(* IEC 61131-3 sources: SmartHomeNew/snapshots/2026-05-25, 217 files *)

(* ---- E_ALERT_PRIORITY.dut ---- *)
{attribute 'strict'}
TYPE E_ALERT_PRIORITY :
(
    ALERT_PRIORITY_NONE := 0,
    ALERT_PRIORITY_LOW := 1,
    ALERT_PRIORITY_MEDIUM := 2,
    ALERT_PRIORITY_HIGH := 3,
    ALERT_PRIORITY_CRITICAL := 4
) USINT;
END_TYPE

(* ---- E_Modbus_Function.dut ---- *)
TYPE E_Modbus_Function :
(
    MB_NONE := 0,
    MB_FC03_READ_HOLDING_REGISTERS := 3,
    MB_FC04_READ_INPUT_REGISTERS := 4,
    MB_FC06_WRITE_SINGLE_REGISTER := 6,
    MB_FC16_WRITE_MULTIPLE_REGISTERS := 16
);
END_TYPE

(* ---- E_OpenTherm_Error.dut ---- *)
TYPE E_OpenTherm_Error :
(
    OT_ERROR_NONE := 0,
    OT_ERROR_HEARTBEAT_TIMEOUT := 1,
    OT_ERROR_ACK_TIMEOUT := 2,
    OT_ERROR_ADAPTER_FAULT := 3,
    OT_ERROR_COMMUNICATION := 4,
    OT_ERROR_INVALID_RESPONSE := 5
);
END_TYPE

(* ---- E_Rule_Condition_Type.dut ---- *)
{attribute 'strict'}
TYPE E_Rule_Condition_Type :
(
    COND_NONE := 0,
    COND_AIR_TEMP := 1,
    COND_FLOOR_TEMP := 2,
    COND_HUMIDITY := 3,
    COND_CO2 := 4,
    COND_METHANE := 5,
    COND_CO := 6,
    COND_DOOR_WINDOW := 7,
    COND_FLOOD := 8,
    COND_SMOKE := 9,
    COND_MOTION := 10,
    COND_TIME_OF_DAY := 11,
    COND_DAY_OF_WEEK := 12
) USINT;
END_TYPE

(* ---- E_RUNTIME_ADAPTIVE_MODE.dut ---- *)
TYPE E_RUNTIME_ADAPTIVE_MODE : (
    FULL_SEMANTIC_MODE,
    REDUCED_ANALYTICS_MODE,
    SURVIVABILITY_MODE,
    MINIMAL_SAFE_MODE
);
END_TYPE

(* ---- E_RUNTIME_TRANSITION_RESULT.dut ---- *)
TYPE E_RUNTIME_TRANSITION_RESULT : (
    TRANSITION_VALID,
    TRANSITION_FORBIDDEN,
    TRANSITION_REQUIRES_PROOF,
    TRANSITION_REQUIRES_RECOVERY,
    TRANSITION_REQUIRES_TEMPORAL_ALIGNMENT
);
END_TYPE

(* ---- E_SCENARIO_TYPE.dut ---- *)
{attribute 'strict'}
TYPE E_SCENARIO_TYPE :
(
    SCENARIO_NONE := 0,
    SCENARIO_MORNING := 1,
    SCENARIO_EVENING := 2,
    SCENARIO_AWAY := 3,
    SCENARIO_PARTY := 4,
    SCENARIO_SLEEP := 5,
    SCENARIO_EMERGENCY := 6,
    SCENARIO_PRESENCE := 7
) USINT;
END_TYPE

(* ---- GVL_CANONICAL_RUNTIME_FABRIC_REGISTRY.gvl ---- *)
TYPE E_GOVERNANCE_PRIORITY_TIER : (
    TIER_0_SAFETY,
    TIER_1_AUTHORITY,
    TIER_2_PHYSICAL_TRUTH,
    TIER_3_SURVIVABILITY,
    TIER_4_OBSERVABILITY,
    TIER_5_ANALYTICS
);
END_TYPE

VAR_GLOBAL
    // Canonical semantic registry.
    Runtime_Fabric_Registry_Active : BOOL := TRUE;
    Runtime_Fabric_Registry_ReadOnly : BOOL := TRUE;

    // Tier hierarchy.
    Current_Governance_Priority_Tier : E_GOVERNANCE_PRIORITY_TIER := TIER_0_SAFETY;

    Tier0_Safety_Active : BOOL := TRUE;
    Tier1_Authority_Active : BOOL := TRUE;
    Tier2_Physical_Truth_Active : BOOL := TRUE;
    Tier3_Survivability_Active : BOOL := TRUE;
    Tier4_Observability_Active : BOOL := TRUE;
    Tier5_Analytics_Active : BOOL := TRUE;

    // Canonical semantic domains.
    Temporal_Integrity_Cluster_Active : BOOL := TRUE;
    Authority_Integrity_Cluster_Active : BOOL := TRUE;
    Physical_Reality_Cluster_Active : BOOL := TRUE;
    Operational_Intelligence_Cluster_Active : BOOL := TRUE;
    Survivability_Cluster_Active : BOOL := TRUE;

    // Runtime compression observations.
    Governance_Scattering_Observed : BOOL := FALSE;
    Semantic_Duplication_Observed : BOOL := FALSE;
    Runtime_Complexity_Pressure_Observed : BOOL := FALSE;

    // Semantic recursion prevention.
    Governance_Depth_Limit_Reached : BOOL := FALSE;
    Semantic_Recursion_Limit_Reached : BOOL := FALSE;
    Verification_Chaining_Limit_Reached : BOOL := FALSE;
    Observability_Amplification_Limit_Reached : BOOL := FALSE;

    // Runtime cost awareness.
    Governance_Runtime_Cost_Observed : BOOL := FALSE;
    Verification_Induced_Instability_Risk : BOOL := FALSE;

    Runtime_Fabric_Registry_Epoch : UDINT := 0;
END_VAR

(* ---- ST_Alarm_Record.dut ---- *)
{attribute 'pack_mode' := '1'}
TYPE ST_Alarm_Record :
STRUCT
    ID : UDINT; // Уникальный идентификатор тревоги
    Timestamp_MS : UDINT; // Время возникновения
    Source : STRING(20); // Источник (Gas, Fire, Flood, Security, System)
    Source_ID : BYTE; // Идентификатор источника (например, номер котла)
    Message : STRING(100); // Описание тревоги
    Severity : E_ALERT_PRIORITY; // Приоритет тревоги
    Is_Active : BOOL; // Тревога все еще активна
    Is_Acknowledged : BOOL; // Квитирована оператором
END_STRUCT
END_TYPE

(* ---- ST_Behavior_Weights.dut ---- *)
TYPE ST_Behavior_Weights :
STRUCT
    W_Comfort : REAL;
    W_Night : REAL;
    W_Preheat : REAL;
    W_VentBoost : REAL;
    W_AccessSecure : REAL;
END_STRUCT
END_TYPE

(* ---- ST_Calibration_Sensor_Summary.dut ---- *)
{attribute 'pack_mode' := '1'}
TYPE ST_Calibration_Sensor_Summary :
STRUCT
    active : BOOL;
    status : INT; // 0=OK,1=IN_PROGRESS,2=WARNING,3=ERROR
    calibrated_value : REAL;
    deviation_percent : REAL;
    verification_active : BOOL;
    verification_failed : BOOL;
    record_index : INT;
    label : STRING(64);
    summary_text : STRING(160);
END_STRUCT
END_TYPE

(* ---- ST_Distributed_Authority_State.dut ---- *)
TYPE ST_Distributed_Authority_State :
STRUCT
    Runtime_Valid : BOOL;
    Runtime_System_Time_MS : UDINT;

    Controller_Id : UINT;
    Runtime_Node_Id : UINT;
    Authority_Domain_Id : UINT;

    Authority_Election_Active : BOOL;
    Authority_Master_Elected : BOOL;
    Authority_Backup_Elected : BOOL;
    Authority_Observer_Only : BOOL;

    Authority_Lease_Valid : BOOL;
    Authority_Lease_Expired : BOOL;
    Authority_Lease_Timeout_MS : UDINT;

    Replication_Consensus_Healthy : BOOL;
    Replication_Consensus_Stale : BOOL;

    Recovery_Authority_Allowed : BOOL;
    Rollback_Authority_Allowed : BOOL;
    Quarantine_Authority_Allowed : BOOL;

    Split_Brain_Blocked : BOOL;
    Distributed_Safety_Barrier_OK : BOOL;

    Status_Code : UINT;
    Status_Text : STRING(160);
END_STRUCT
END_TYPE

(* ---- ST_Distributed_Orchestration_State.dut ---- *)
TYPE ST_Distributed_Orchestration_State :
STRUCT
    Runtime_Valid : BOOL;
    Runtime_System_Time_MS : UDINT;

    Orchestration_Sequence_Id : UDINT;
    Distributed_Execution_Active : BOOL;

    Cross_Node_Isolation_Required : BOOL;
    Cross_Node_Recovery_Required : BOOL;
    Cross_Node_Rollback_Required : BOOL;

    Distributed_Projection_Granted : BOOL;
    Distributed_Projection_Blocked : BOOL;

    Distributed_Rollback_Allowed : BOOL;
    Distributed_Recovery_Allowed : BOOL;

    Distributed_Scheduler_Healthy : BOOL;
    Distributed_Timing_Window_Valid : BOOL;

    Remote_Node_Ack_Required : BOOL;
    Remote_Node_Ack_Received : BOOL;

    Distributed_Conflict_Detected : BOOL;
    Distributed_Split_Execution_Suspected : BOOL;

    Status_Code : UINT;
    Status_Text : STRING(160);
END_STRUCT
END_TYPE

(* ---- ST_Flood_Global_Config.dut ---- *)
{attribute 'pack_mode' := '1'}
TYPE ST_Flood_Global_Config :
STRUCT
    // Isolation groups:
    // 1 = стояк 1 кухня, 2 = стояк 2 мастер-санузел,
    // 3 = стояк 3 гостевые санузлы + постирочная,
    // 4 = общий ввод ХВС/ГВС, legacy chains 35/36.
    // Вода от скважины: при потере питания насос останавливается и давления нет,
    // поэтому базовая эксплуатационная модель — нормально-открытые краны с
    // электроприводом и концевиками, закрываемые при аварии.
    valve_types : ARRAY[1..GVL_CONSTANTS.C_MAX_FLOOD_VALVES] OF E_VALVE_TYPE := [GVL_CONSTANTS.C_MAX_FLOOD_VALVES(E_VALVE_TYPE.VALVE_NO)];

    // 1-2 кухня -> стояк 1;
    // 3-4 мастер-санузел -> стояк 2;
    // 5-9 гостевые санузлы + постирочная -> стояк 3;
    // 10-12 котельная/ХВП/общий ввод -> общий ввод 35/36.
    sensor_to_valve_map : ARRAY[1..GVL_CONSTANTS.C_MAX_FLOOD_SENSORS] OF BYTE := [1, 1, 2, 2, 3, 3, 3, 3, 3, 4, 4, 4];

    min_duration_ms : UDINT := 5000; // Защита от брызг (5 сек)
    warning_duration_ms : UDINT := 30000; // Время предупреждения до перекрытия (30 сек)
END_STRUCT
END_TYPE

(* ---- ST_FloorHeating_Circuit_Config.dut ---- *)
{attribute 'pack_mode' := '1'}
TYPE ST_FloorHeating_Circuit_Config :
STRUCT
    circuit_id : BYTE := 0;
    zone : BYTE := 0;
    manifold_id : BYTE := 1; // ID коллектора, к которому подключен контур
    sensor_id : BYTE := 1; // ID датчика температуры
    valve_id : BYTE := 1; // ID клапана
    control_type : BYTE := 1; // 0: по полу, 1: по воздуху

    // Legacy/default setpoint. Kept for backward compatibility.
    // If comfort_temp <= 0.0, design_temp remains the comfort setpoint.
    design_temp : REAL := 35.0;

    // Per-room/per-circuit comfort and economy policy.
    // use_in_normal=FALSE keeps the circuit at economy_temp even in normal mode.
    // use_in_away_preheat=TRUE allows planned-return preheat to comfort_temp.
    use_in_normal : BOOL := TRUE;
    use_in_away_preheat : BOOL := TRUE;
    comfort_temp : REAL := 0.0; // 0.0 = use design_temp
    economy_temp : REAL := 16.0;
    long_away_temp : REAL := 12.0;

    min_temp : REAL := 20.0;
    max_temp : REAL := 45.0;
    pid_kp : REAL := 2.0;
    pwm_period_s : UINT := 600; // Период ШИМ в секундах (по умолчанию 10 минут)
END_STRUCT
END_TYPE

(* ---- ST_Forensic_Journal_Record.dut ---- *)
TYPE ST_Forensic_Journal_Record :
STRUCT
    Record_Valid : BOOL;
    Event_Time_MS : UDINT;
    Event_Id : UDINT;
    Event_Class : UINT;
    Event_Severity : UINT;

    Config_Version : UDINT;
    Topology_Version : UDINT;
    Recovery_Domain_Id : UINT;
    Valve_Group_Id : UINT;
    Sensor_Id : UINT;

    Activation_Event : BOOL;
    Rollback_Event : BOOL;
    Quarantine_Event : BOOL;
    Recovery_Event : BOOL;
    Restart_Event : BOOL;

    Status_Code : UINT;
    Event_Text : STRING(160);
END_STRUCT
END_TYPE

(* ---- ST_Heating_Circuit_Runtime_Projection.dut ---- *)
TYPE ST_Heating_Circuit_Runtime_Projection :
STRUCT
    // Passive runtime-to-observability projection contract.
    // Contains semantic runtime state only.
    // No runtime authority.

    Visible : BOOL;

    // Selected operational source
    Selected_Source_Code : UINT; // 0 none, 1 room, 2 floor
    Selected_Source_Confidence : REAL;

    // Runtime degraded semantics
    Fallback_Active : BOOL;
    Source_Degraded : BOOL;
    Sensor_Error_Active : BOOL;

    // Explainability semantics
    Reason_Code : UINT;
    Reason_Text : STRING(128);

    // Runtime semantic edge publication
    Source_Switched_Event : BOOL;
    Fallback_Activated_Event : BOOL;
    Fallback_Recovered_Event : BOOL;
    Source_Loss_Event : BOOL;

    Last_Event_Code : UINT;
    Last_Event_Text : STRING(128);
    Last_Event_MS : UDINT;
END_STRUCT
END_TYPE

(* ---- ST_Heating_Runtime_Blackbox_Timeline.dut ---- *)
TYPE ST_Heating_Runtime_Blackbox_Timeline :
STRUCT
    // ======================================================
    // Blackbox events
    // ======================================================
    Events : ARRAY[1..256] OF ST_Heating_Runtime_Blackbox_Event;

    // ======================================================
    // Timeline state
    // ======================================================
    Write_Index : UINT;
    Event_Count : UINT;
    Timeline_Overflow : BOOL;

    // ======================================================
    // Runtime forensic state
    // Passive forensic visibility only.
    // No replay activation authority exists.
    // ======================================================
    Reconstruction_Visible : BOOL;
    Forensic_Timeline_Visible : BOOL;
    Root_Cause_Reconstructed : BOOL;

    // ======================================================
    // Timeline integrity
    // ======================================================
    Sequencing_Valid : BOOL;
    Ownership_Valid : BOOL;
    Synchronization_Valid : BOOL;

    // ======================================================
    // Timeline status
    // ======================================================
    Status_Code : UINT;
    Status_Text : STRING(128);
END_STRUCT
END_TYPE

(* ---- ST_Heating_Runtime_Context.dut ---- *)
TYPE ST_Heating_Runtime_Context :
STRUCT
    // ======================================================
    // Runtime lifecycle
    // ======================================================
    Runtime_Enabled : BOOL;
    Runtime_Ready : BOOL;
    Runtime_Fault : BOOL;

    // ======================================================
    // Runtime phase model
    // ======================================================
    Current_Phase : E_Heating_Runtime_Phase;

    // ======================================================
    // Phase execution permissions
    // ======================================================
    Allow_DHW_Phase : BOOL;
    Allow_Heating_Phase : BOOL;
    Allow_Service_Gating_Phase : BOOL;
    Allow_State_Publication_Phase : BOOL;
    Allow_Diagnostics_Phase : BOOL;
    Allow_Output_Projection_Phase : BOOL;

    // ======================================================
    // Runtime sequencing validation
    // ======================================================
    DHW_Executed : BOOL;
    Heating_Executed : BOOL;
    Service_Gating_Executed : BOOL;
    State_Publication_Executed : BOOL;
    Diagnostics_Executed : BOOL;
    Output_Projection_Executed : BOOL;

    // ======================================================
    // Runtime ordering integrity
    // ======================================================
    DHW_Before_Heating_Valid : BOOL;
    State_Publication_Before_Diagnostics_Valid : BOOL;
    Output_Projection_Last_Valid : BOOL;

    // ======================================================
    // Runtime status
    // ======================================================
    Runtime_Status_Code : UINT;
    Runtime_Status_Text : STRING(128);

    // ======================================================
    // Diagnostics / explainability isolation
    // ======================================================
    Diagnostics_Isolation_Valid : BOOL;
    Explainability_Isolation_Valid : BOOL;

    // ======================================================
    // Safety isolation
    // ======================================================
    Safety_Isolation_Valid : BOOL;

    // ======================================================
    // OpenTherm ownership isolation
    // ======================================================
    OpenTherm_Ownership_Valid : BOOL;

    // ======================================================
    // Cascade ownership isolation
    // ======================================================
    Cascade_Ownership_Valid : BOOL;
END_STRUCT
END_TYPE

(* ---- ST_Heating_Runtime_Observation.dut ---- *)
TYPE ST_Heating_Runtime_Observation :
STRUCT
    // ======================================================
    // Runtime execution state
    // ======================================================
    Runtime_Active : BOOL;
    Runtime_Ready : BOOL;
    Runtime_Fault : BOOL;

    // ======================================================
    // Runtime phase observation
    // ======================================================
    Current_Phase : E_Heating_Runtime_Phase;

    // ======================================================
    // DHW runtime observation
    // ======================================================
    DHW_Demand_Active : BOOL;
    DHW_Heating_Active : BOOL;
    DHW_Circulation_Active : BOOL;

    // ======================================================
    // Heating runtime observation
    // ======================================================
    Heating_Demand_Active : BOOL;
    Heating_Runtime_Active : BOOL;
    Heating_Output_Active : BOOL;

    // ======================================================
    // Cascade runtime observation
    // ======================================================
    Cascade_Available : BOOL;
    Cascade_Degraded : BOOL;
    Cascade_Active_Boilers : UINT;
    Cascade_Available_Boilers : UINT;

    // ======================================================
    // OpenTherm runtime observation
    // ======================================================
    OpenTherm_Online : BOOL;
    OpenTherm_Command_Valid : BOOL;
    OpenTherm_Transport_Degraded : BOOL;

    // ======================================================
    // Diagnostics observation
    // ======================================================
    Diagnostics_Active : BOOL;
    Explainability_Active : BOOL;

    // ======================================================
    // Runtime sequencing observation
    // ======================================================
    DHW_Before_Heating_Observed : BOOL;
    Diagnostics_After_Publication_Observed : BOOL;
    Output_Projection_Last_Observed : BOOL;

    // ======================================================
    // Runtime ownership observation
    // ======================================================
    Runtime_Ownership_Valid : BOOL;
    Diagnostics_Ownership_Valid : BOOL;
    OpenTherm_Ownership_Valid : BOOL;
    Cascade_Ownership_Valid : BOOL;
    Safety_Ownership_Valid : BOOL;

    // ======================================================
    // Runtime observation status
    // ======================================================
    Observation_Status_Code : UINT;
    Observation_Status_Text : STRING(128);
END_STRUCT
END_TYPE

(* ---- ST_Heating_Runtime_Phase_Transition.dut ---- *)
TYPE ST_Heating_Runtime_Phase_Transition :
STRUCT
    // ======================================================
    // Phase transition state
    // ======================================================
    Previous_Phase : E_Heating_Runtime_Phase;
    Current_Phase : E_Heating_Runtime_Phase;
    Next_Phase : E_Heating_Runtime_Phase;

    // ======================================================
    // Transition lifecycle
    // ======================================================
    Transition_Active : BOOL;
    Transition_Completed : BOOL;
    Transition_Failed : BOOL;

    // ======================================================
    // Transition timing
    // ======================================================
    Transition_Start_MS : UDINT;
    Transition_End_MS : UDINT;
    Transition_Duration_MS : UDINT;

    // ======================================================
    // Transition integrity
    // ======================================================
    Sequencing_Valid : BOOL;
    Ownership_Valid : BOOL;
    Synchronization_Valid : BOOL;

    // ======================================================
    // Transition status
    // ======================================================
    Status_Code : UINT;
    Status_Text : STRING(128);
END_STRUCT
END_TYPE

(* ---- ST_IO_Binding_Record.dut ---- *)
TYPE ST_IO_Binding_Record :
STRUCT
    Binding_Valid : BOOL;
    Binding_Version : UDINT;

    Physical_Channel_Id : UINT;
    Logical_Device_Id : UINT;
    Domain_Id : UINT;
    Role_Id : UINT;

    Controller_Id : UINT;
    Module_Id : UINT;
    Terminal_Id : UINT;

    Inverted : BOOL;
    Required : BOOL;
    Quality_Required : BOOL;

    Status_Code : UINT;
    Status_Text : STRING(128);
END_STRUCT
END_TYPE

(* ---- ST_Modbus_Request.dut ---- *)
TYPE ST_Modbus_Request :
STRUCT
    Enable : BOOL;
    Slave_ID : BYTE;
    Function_Code : E_Modbus_Function;
    Start_Register : UINT;
    Register_Count : UINT;
    Write_Value : ARRAY[1..32] OF WORD;
    Sequence : UDINT;
    Timeout_MS : UDINT;
END_STRUCT
END_TYPE

(* ---- ST_OpenTherm_Command.dut ---- *)
TYPE ST_OpenTherm_Command :
STRUCT
    Enable : BOOL;
    Setpoint_x10 : UINT;
    Sequence : UDINT;
    Last_Write_MS : UDINT;
END_STRUCT
END_TYPE

(* ---- ST_OpenTherm_Wire_Image.dut ---- *)
TYPE ST_OpenTherm_Wire_Image :
STRUCT
    // Command image to be written to the physical adapter.
    Cmd_Enable : WORD;
    Cmd_Setpoint_x10 : WORD;
    Cmd_Seq_Lo : WORD;
    Cmd_Seq_Hi : WORD;

    // Status image read from the physical adapter.
    Status_Heartbeat_Lo : WORD;
    Status_Heartbeat_Hi : WORD;
    Status_Ack_Seq_Lo : WORD;
    Status_Ack_Seq_Hi : WORD;
    Status_Word : WORD;
    Error_Code : WORD;
    Modulation_x10 : WORD;
    Boiler_Temp_x10 : WORD;
END_STRUCT
END_TYPE

(* ---- ST_Runtime_Node_Discovery_State.dut ---- *)
TYPE ST_Runtime_Node_Discovery_State :
STRUCT
    Runtime_Valid : BOOL;
    Runtime_System_Time_MS : UDINT;

    Discovery_Active : BOOL;
    Node_Discovered : BOOL;
    Node_Validated : BOOL;
    Node_Authorized : BOOL;
    Node_Quarantined : BOOL;

    Controller_Id : UINT;
    Runtime_Node_Id : UINT;
    Authority_Class : UINT;

    Deployment_Assigned : BOOL;
    Execution_Domain_Assigned : BOOL;
    Capability_Validated : BOOL;

    Discovery_Timeout : BOOL;
    Discovery_Rejected : BOOL;

    Status_Code : UINT;
    Status_Text : STRING(160);
END_STRUCT
END_TYPE

(* ---- ST_System_State_Summary.dut ---- *)
{attribute 'pack_mode' := '1'}
TYPE ST_System_State_Summary :
STRUCT
    Outdoor_Temp : REAL;
    Indoor_Temp : ARRAY[1..GVL_CONSTANTS.C_MAX_CLIMATE_ZONES] OF REAL;
    Floor_Temps : ARRAY[1..GVL_CONSTANTS.C_MAX_HEATING_CIRCUITS] OF REAL;
    Humidity : ARRAY[1..GVL_CONSTANTS.C_MAX_HUMIDITY_SENSORS] OF REAL;
    CO2 : ARRAY[1..GVL_CONSTANTS.C_MAX_CO2_SENSORS] OF REAL;
    Gas_Alarm : BOOL;
    Flood_Alarm : BOOL;
    Fire_Alarm : BOOL;
    Security_Alarm : BOOL;
    Security_Armed : BOOL;
END_STRUCT
END_TYPE

(* ---- ST_Tariff_Config.dut ---- *)
{attribute 'pack_mode' := '1'}
TYPE ST_Tariff_Config :
STRUCT
    Enabled : BOOL := FALSE;
    Night_Start_Hour : UINT := 23;
    Night_End_Hour : UINT := 7;
    Boost_Delta : REAL := 2.0;
END_STRUCT
END_TYPE

(* ---- ST_Ventilation_Scenario_Mode.dut ---- *)
{attribute 'pack_mode' := '1'}
TYPE ST_Ventilation_Scenario_Mode :
STRUCT
  Scenario_ID : BYTE;
  Scenario_Priority : BYTE;
  Fire_Alarm : BOOL;
  Methane_Alarm : BOOL;
  Smoke_Detected : BOOL;
  Exhaust_Modes : ARRAY[1..GVL_CONSTANTS.C_MAX_EXHAUST_FANS] OF BYTE;
  Supply_Modes : ARRAY[1..GVL_CONSTANTS.C_MAX_SUPPLY_FANS] OF BYTE;
  Base_Fan_Speed : BYTE := 50;
  Target_Temp : REAL := 22.0;
END_STRUCT
END_TYPE

(* ---- ST_Water_Graph_Traversal_State.dut ---- *)
TYPE ST_Water_Graph_Traversal_State :
STRUCT
    Runtime_Valid : BOOL;
    Runtime_System_Time_MS : UDINT;

    Sensor_Id : UINT;
    Start_Segment_Id : UINT;
    Target_Valve_Group_Id : UINT;

    Upstream_Dependency_Detected : BOOL;
    Downstream_Impact_Detected : BOOL;
    Shared_Trunk_Traversal : BOOL;

    Traversal_Valid : BOOL;
    Traversal_Conflict : BOOL;
    Traversal_Ambiguous : BOOL;

    Dependency_Depth : UINT;

    Selective_Path_Allowed : BOOL;
    Global_Fallback_Required : BOOL;

    Status_Code : UINT;
    Status_Text : STRING(128);
END_STRUCT
END_TYPE

(* ---- ST_Water_Isolation_Authority_State.dut ---- *)
TYPE ST_Water_Isolation_Authority_State :
STRUCT
    // ==============================================================================
    // Water/Flood isolation authority decision state.
    // ==============================================================================
    //
    // Deterministic authority-candidate contract.
    // This contract does NOT directly write physical outputs.
    // Final output ownership remains in command arbitration/output projection.
    // ==============================================================================

    Decision_Valid : BOOL;
    Decision_System_Time_MS : UDINT;

    // Requested authority.
    Isolation_Requested : BOOL;
    Selective_Candidate : BOOL;
    Global_Fallback_Candidate : BOOL;

    // Authority decision.
    Selective_Authority_Allowed : BOOL;
    Global_Fallback_Required : BOOL;
    Authority_Denied : BOOL;

    // Deterministic target.
    Hydraulic_Zone_Id : UINT;
    Isolation_Group_Id : UINT;
    Valve_Group_Id : UINT;

    // Validation inputs.
    Mapping_Valid : BOOL;
    Deterministic_Target_Valid : BOOL;
    Safety_Context_Allows_Selective : BOOL;
    Valve_Diagnostics_Available : BOOL;
    Valve_Confirmation_Required : BOOL;

    // Runtime compatibility visibility.
    Active_Global_Close_Path : BOOL;
    Active_Safety_Latch : BOOL;

    // Explainability.
    Decision_Code : UINT;
    Decision_Text : STRING(128);

    // Lifecycle edges.
    Authority_Selected_Event : BOOL;
    Authority_Denied_Event : BOOL;
    Fallback_Selected_Event : BOOL;
END_STRUCT
END_TYPE

(* ---- ST_Water_Isolation_Path_Runtime_State.dut ---- *)
TYPE ST_Water_Isolation_Path_Runtime_State :
STRUCT
    Runtime_Valid : BOOL;
    Runtime_System_Time_MS : UDINT;

    Sensor_Id : UINT;

    Isolation_Path_Valid : BOOL;
    Isolation_Path_Ambiguous : BOOL;
    Multi_Valve_Path : BOOL;

    Active_Isolation_Group_Id : UINT;
    Active_Valve_Group_Id : UINT;

    Shared_Trunk_Impact : BOOL;
    Cross_Zone_Impact : BOOL;

    Selective_Isolation_Allowed : BOOL;
    Global_Fallback_Required : BOOL;

    Conflict_Detected : BOOL;

    Status_Code : UINT;
    Status_Text : STRING(128);
END_STRUCT
END_TYPE

(* ---- ST_Water_Output_Projection_State.dut ---- *)
TYPE ST_Water_Output_Projection_State :
STRUCT
    // Deterministic output projection contract.

    Projection_Valid : BOOL;
    Projection_System_Time_MS : UDINT;

    // Ownership.
    Output_Owner_Valid : BOOL;
    Output_Owner_Id : UINT;

    // Projection target.
    Valve_Id : UINT;
    Valve_Group_Id : UINT;

    // Authority source.
    Selective_Authority_Allowed : BOOL;
    Global_Fallback_Required : BOOL;
    Authority_Valid : BOOL;

    // Physical projection.
    Physical_Close_Project : BOOL;
    Physical_Open_Project : BOOL;

    // Reconciliation hooks.
    Expected_Closed : BOOL;
    Expected_Open : BOOL;
    Confirmed_Closed : BOOL;
    Confirmed_Open : BOOL;
    Confirmation_Unknown : BOOL;

    // Arbitration validity.
    Projection_Allowed : BOOL;
    Projection_Denied : BOOL;

    // Explainability.
    Projection_Code : UINT;
    Projection_Text : STRING(128);

    // Lifecycle.
    Projection_Activated_Event : BOOL;
    Projection_Denied_Event : BOOL;
END_STRUCT
END_TYPE

(* ---- ST_Water_Recovery_FSM_State.dut ---- *)
TYPE ST_Water_Recovery_FSM_State :
STRUCT
    Runtime_Valid : BOOL;
    Runtime_System_Time_MS : UDINT;

    Recovery_Domain_Id : UINT;

    Recovery_Requested : BOOL;
    Recovery_Sequencing_Active : BOOL;
    Recovery_Verification_Window_Active : BOOL;

    Rollback_Required : BOOL;
    Escalation_Required : BOOL;
    Operator_Ack_Required : BOOL;

    Recovery_Completed : BOOL;
    Recovery_Denied : BOOL;

    FSM_State : UINT;

    Status_Code : UINT;
    Status_Text : STRING(128);
END_STRUCT
END_TYPE

(* ---- ST_Water_Topology_Config_Record.dut ---- *)
TYPE ST_Water_Topology_Config_Record :
STRUCT
    Config_Valid : BOOL;
    Config_Version : UDINT;

    Sensor_Id : UINT;
    Logical_Zone_Id : UINT;
    Hydraulic_Segment_Id : UINT;
    Isolation_Group_Id : UINT;
    Primary_Valve_Group_Id : UINT;
    Secondary_Valve_Group_Id : UINT;
    Fallback_Domain_Id : UINT;

    Shared_Trunk : BOOL;
    Cross_Zone_Dependency : BOOL;
    Multi_Valve_Required : BOOL;

    Recovery_Domain_Id : UINT;
    Recovery_Requires_Manual_Ack : BOOL;

    Status_Code : UINT;
    Status_Text : STRING(128);
END_STRUCT
END_TYPE

(* ---- ST_Water_Valve_Feedback_State.dut ---- *)
TYPE ST_Water_Valve_Feedback_State :
STRUCT
    Runtime_Valid : BOOL;
    Runtime_System_Time_MS : UDINT;

    Valve_Group_Id : UINT;

    Feedback_Available : BOOL;

    Physical_Open_Feedback : BOOL;
    Physical_Closed_Feedback : BOOL;

    Confirmed_Open : BOOL;
    Confirmed_Closed : BOOL;
    Confirmation_Unknown : BOOL;

    Feedback_Invalid : BOOL;
    Feedback_Conflict : BOOL;
    Feedback_Timeout : BOOL;

    Travel_Timeout_Active : BOOL;
    Valve_Stuck_Suspected : BOOL;

    Valve_Degraded : BOOL;

    Status_Code : UINT;
    Status_Text : STRING(128);
END_STRUCT
END_TYPE

(* ---- ST_Water_Valve_Runtime_State.dut ---- *)
TYPE ST_Water_Valve_Runtime_State :
STRUCT
    // ==============================================================================
    // Water/Flood valve runtime semantic state.
    // ==============================================================================
    //
    // Observe-first valve governance contract.
    //
    // This contract does NOT directly own physical outputs.
    // ==============================================================================

    Runtime_Valid : BOOL;
    Runtime_System_Time_MS : UDINT;

    // Valve identity.
    Valve_Id : UINT;
    Valve_Group_Id : UINT;

    // Authority/runtime semantics.
    Close_Requested : BOOL;
    Open_Requested : BOOL;
    Global_Fallback_Request : BOOL;
    Selective_Authority_Allowed : BOOL;

    // Output/runtime visibility.
    Physical_Output_Active : BOOL;
    Output_Command_Projected : BOOL;

    // Confirmation semantics.
    Confirmation_Available : BOOL;
    Confirmed_Open : BOOL;
    Confirmed_Closed : BOOL;
    Confirmation_Timeout : BOOL;
    Confirmation_Unknown : BOOL;

    // Diagnostics.
    Diagnostics_Available : BOOL;
    Valve_Healthy : BOOL;
    Valve_Stuck_Suspected : BOOL;
    Travel_Time_Degraded : BOOL;
    Current_Deviation_Detected : BOOL;

    // Governance/degraded semantics.
    Valve_Degraded : BOOL;
    Unsafe_Reopen_Denied : BOOL;
    Recovery_Allowed : BOOL;

    // Explainability.
    Status_Code : UINT;
    Status_Text : STRING(128);

    // Lifecycle edges.
    Close_Command_Event : BOOL;
    Open_Command_Event : BOOL;
    Confirmation_Lost_Event : BOOL;
    Valve_Degraded_Event : BOOL;
END_STRUCT
END_TYPE

(* ---- GVL_ACCESS_RUNTIME.gvl ---- *)
{attribute 'qualified_only'}
VAR_GLOBAL
    // Access domain execution feedback. Observational only.

    G_Runtime_Required : BOOL := FALSE;
    G_Runtime_Executed : BOOL := FALSE;
    G_Runtime_Idle_By_Design : BOOL := FALSE;
    G_Runtime_Blocked_By_Distributed_Gates : BOOL := FALSE;
    G_Any_Pulse_Active : BOOL := FALSE;
    G_Last_Update_MS : UDINT := 0;
    G_Status_Code : UINT := 0;
    G_Status_Text : STRING(128) := '';
END_VAR

(* ---- GVL_ACTUATION_AUTHORITY.gvl ---- *)
VAR_GLOBAL
    // Global actuation authority.
    Actuation_Authority_Valid : BOOL := FALSE;
    Actuation_Authority_Granted : BOOL := FALSE;
    Actuation_Quarantine_Active : BOOL := TRUE;

    // Deterministic actuation epochs.
    Actuation_Command_Epoch : UDINT := 0;
    Field_ACK_Epoch : UDINT := 0;
    Actuation_Authority_Epoch : UDINT := 0;

    // Field-confirmed execution.
    Field_Device_ACK_Valid : BOOL := FALSE;
    Actuator_Transition_Observed : BOOL := FALSE;
    Physical_Convergence_Confirmed : BOOL := FALSE;
    Stable_Physical_Convergence : BOOL := FALSE;

    // Physical execution validation.
    Current_Signature_Confirmed : BOOL := FALSE;
    Flow_Response_Confirmed : BOOL := FALSE;
    Pressure_Response_Confirmed : BOOL := FALSE;
    Motion_Response_Confirmed : BOOL := FALSE;

    // Failure/replay/skew detection.
    Stale_Field_ACK_Detected : BOOL := FALSE;
    Write_Without_Confirm_Detected : BOOL := FALSE;
    Relay_Weld_Suspected : BOOL := FALSE;
    Actuator_Stall_Detected : BOOL := FALSE;
    Partial_Actuation_Detected : BOOL := FALSE;
    Command_Actuation_Skew_Detected : BOOL := FALSE;
    ACK_Replay_Suspected : BOOL := FALSE;

    // Temporal authority.
    Actuation_Last_Update_MS : UDINT := 0;
    Actuation_Lease_Expired : BOOL := TRUE;

    // Diagnostics.
    Actuation_Last_Error_Code : UDINT := 0;
    Actuation_Last_Error_Text : STRING(160) := '';
    Actuation_Invalidation_Count : UDINT := 0;
END_VAR

(* ---- GVL_AUTHORITY_RESURRECTION_BOUNDARY_FABRIC.gvl ---- *)
VAR_GLOBAL
    Authority_Resurrection_Boundary_Valid : BOOL := FALSE;
    Authority_Resurrection_Bounded : BOOL := FALSE;
    Authority_Recovery_Lineage_Stable : BOOL := FALSE;
    Distributed_Authority_Recovery_Consensus : BOOL := FALSE;

    Authority_Resurrection_Causality_Valid : BOOL := FALSE;
    Resurrection_Timeline_Monotonic : BOOL := FALSE;

    Partial_Recovery_Authority_Leak : BOOL := FALSE;
    Unsafe_Authority_Resurrection_Detected : BOOL := FALSE;
    Resurrection_Authority_Fork_Detected : BOOL := FALSE;

    Authority_Resurrection_Epoch : UDINT := 0;
END_VAR

(* ---- GVL_AWAY_HEATING_HMI.gvl ---- *)
{attribute 'qualified_only'}
VAR_GLOBAL
    // HMI surface for per-circuit comfort/economy/away heating profile.
    G_Set_Circuit_Profile_Req : BOOL := FALSE;
    G_Profile_Circuit : INT := 0;
    G_Profile_Use_In_Normal : BOOL := TRUE;
    G_Profile_Use_In_Away_Preheat : BOOL := TRUE;
    G_Profile_Comfort_Temp : REAL := 22.0;
    G_Profile_Economy_Temp : REAL := 17.0;
    G_Profile_Long_Away_Temp : REAL := 12.0;

    // HMI surface for planned return.
    // Delay is relative to current monotonic PLC time, in hours.
    G_Set_Planned_Return_Req : BOOL := FALSE;
    G_Clear_Planned_Return_Req : BOOL := FALSE;
    G_Planned_Return_Enabled : BOOL := FALSE;
    G_Planned_Return_Delay_Hours : REAL := 0.0;
    G_Preheat_Lead_Hours : REAL := 3.0;
    G_Return_Grace_Hours : REAL := 24.0;

    G_Last_Status_Text : STRING(200) := '';
    G_Last_Error : BOOL := FALSE;
    G_Last_Update_MS : UDINT := 0;
END_VAR

(* ---- GVL_CAUSALITY_REVERSAL_PREVENTION_FABRIC.gvl ---- *)
VAR_GLOBAL
    Causality_Reversal_Prevention_Valid : BOOL := FALSE;
    Causality_Reversal_Prevention_Granted : BOOL := FALSE;

    Causality_Reversal_Prevented : BOOL := FALSE;
    Authority_Ordering_Canonical : BOOL := FALSE;
    Revocation_Resurrection_Boundary_Stable : BOOL := FALSE;

    Reversal_Causality_Grounded : BOOL := FALSE;
    Distributed_Reversal_Consensus_Valid : BOOL := FALSE;

    Causality_Reversal_Detected : BOOL := FALSE;
    Resurrection_After_Revocation_Detected : BOOL := FALSE;
    Unsafe_Temporal_Replay_Detected : BOOL := FALSE;

    Causality_Reversal_Epoch : UDINT := 0;
END_VAR

(* ---- GVL_COMMAND_ARBITRATION_BUFFER.gvl ---- *)
{attribute 'qualified_only'}
VAR_GLOBAL
    // Deterministic command arbitration buffer.
    // Owned by PRG_Command_Arbitration and its phase programs only.

    B_Mode : E_Safety_Mode := NORMAL;
    B_Safety_Active : BOOL := FALSE;
    B_User_Access_OK : BOOL := FALSE;

    B_Role_Conflict_Active : BOOL := FALSE;
    B_PLC_Inactive_Active : BOOL := FALSE;

    B_Gas_Valve_Close : BOOL := FALSE;
    B_Boiler_Stop : BOOL := FALSE;
    B_Supply_100_Req : BOOL := FALSE;
    B_Supply_80_Req : BOOL := FALSE;
    B_Vent_PV3_Boost : BOOL := FALSE;
    B_Exhaust_100_Req : BOOL := FALSE;
    B_Vent_Stop : BOOL := FALSE;
    B_Vent_Block : BOOL := FALSE;
    B_Vent_Smoke_Exhaust : BOOL := FALSE;

    B_Heating_Block : BOOL := FALSE;
    B_Heating_Emergency_Stop : BOOL := FALSE;
    B_Heating_Gas_Safety_Stop : BOOL := FALSE;

    B_Water_Block : BOOL := FALSE;
    B_Water_Emergency_Stop : BOOL := FALSE;
    B_Close_Valve_35 : BOOL := FALSE;
    B_Close_Valve_36 : BOOL := FALSE;

    B_Lock_1_Open : BOOL := FALSE;
    B_Lock_1_Close : BOOL := FALSE;
    B_Lock_2_Open : BOOL := FALSE;
    B_Lock_2_Close : BOOL := FALSE;
    B_Gate_Open : BOOL := FALSE;
    B_Wicket_Open : BOOL := FALSE;
END_VAR

(* ---- GVL_COMMAND_POLICY_CONFIG.gvl ---- *)
{attribute 'qualified_only'}
VAR_GLOBAL
    // Command Arbitration safety policy configuration.
    // Used by PRG_Command_Arbitration only.

    // PLC inactive fail-safe policy.
    G_PLC_Inactive_Close_Gas : BOOL := TRUE;
    G_PLC_Inactive_Stop_Boiler : BOOL := TRUE;
    G_PLC_Inactive_Block_Heating : BOOL := TRUE;
    G_PLC_Inactive_Stop_Vent : BOOL := TRUE;
    G_PLC_Inactive_Block_Water : BOOL := TRUE;

    // FIRE policy.
    G_Fire_Block_Heating : BOOL := TRUE;
    G_Fire_Stop_Boiler : BOOL := TRUE;
    G_Fire_Stop_Vent : BOOL := TRUE;
    G_Fire_Open_Lock_1 : BOOL := TRUE;
    G_Fire_Open_Lock_2 : BOOL := TRUE;
    G_Fire_Open_Gate : BOOL := TRUE;
    G_Fire_Open_Wicket : BOOL := TRUE;
    G_Fire_Block_Lock_Close : BOOL := TRUE;

    // GAS policy.
    G_Gas_Close_Gas : BOOL := TRUE;
    G_Gas_Stop_Boiler : BOOL := TRUE;
    G_Gas_Block_Heating : BOOL := TRUE;
    G_Gas_Open_Gate : BOOL := TRUE;
    G_Gas_Open_Wicket : BOOL := TRUE;
    // Intentionally FALSE by project decision: Lock 1/2 are not evacuation contour for GAS.
    G_Gas_Open_Lock_1 : BOOL := FALSE;
    G_Gas_Open_Lock_2 : BOOL := FALSE;

    // WATER policy.
    G_Water_Block_Water : BOOL := TRUE;

    // GLOBAL_STOP policy.
    G_GlobalStop_Block_Heating : BOOL := TRUE;
    G_GlobalStop_Stop_Boiler : BOOL := TRUE;
    G_GlobalStop_Stop_Vent : BOOL := TRUE;
    G_GlobalStop_Block_Water : BOOL := TRUE;

    // Sanity policy.
    G_Block_Close_When_Open_Commanded : BOOL := TRUE;
END_VAR

(* ---- GVL_COMMAND_VERIFY.gvl ---- *)
VAR_GLOBAL
    Command_Mismatch_Count : INT := 0;
    Command_Match_OK : BOOL := TRUE;
    Command_Mismatch_Active : BOOL := FALSE;

    Runtime_Sanity_OK : BOOL := TRUE;
    Runtime_Sanity_Error_Count : UDINT := 0;
    Runtime_Last_Error_Code : UDINT := 0;
    Runtime_Last_Error_Time_MS : UDINT := 0;
    Runtime_Last_Error_Text : STRING(160) := '';

    PreOutput_Barrier_OK : BOOL := TRUE;
    PreOutput_Block_IO : BOOL := FALSE;
    PreOutput_Physical_Causality_Valid : BOOL := FALSE;
    PreOutput_Block_Count : UDINT := 0;
    PreOutput_Last_Error_Code : UDINT := 0;
    PreOutput_Last_Error_Time_MS : UDINT := 0;
    PreOutput_Last_Error_Text : STRING(160) := '';
END_VAR

(* ---- GVL_CONFIG.gvl ---- *)
{attribute 'qualified_only'}
VAR_GLOBAL
    // Subsystem Configurations
    G_Heating_Config : ST_Heating_Config;
    G_DHW_Config : ST_DHW_Config;
    G_Security_Config : ST_Security_Global_Config;

    // HMI Configurations
    G_HMI_FloorHeating_Configs : ARRAY[1..GVL_CONSTANTS.C_MAX_HEATING_CIRCUITS] OF ST_FloorHeating_Circuit_Config;
    G_Heating_Circuit_To_Zone : ARRAY[1..GVL_CONSTANTS.C_MAX_HEATING_CIRCUITS] OF INT := [1, 2, 3, 4, 5, 6, 7, 8, 9, 10, 11, 12, 13, 14, 15, 16];
    G_Wet_Zone_Map : ARRAY[1..32] OF BOOL;
    G_HMI_Tariff_Settings : ST_Tariff_Config;
    G_HMI_Vent_Global_Config : ST_Ventilation_Global_Config;
    G_HMI_Scenario_Configs : ARRAY[1..GVL_CONSTANTS.C_MAX_SCENARIOS] OF ST_Scenario_Config;
    G_HMI_Flood_Config : ST_Flood_Global_Config;
    G_Flood_Global_Config : ST_Flood_Global_Config;
    G_HMI_User_Rules : ARRAY[1..GVL_CONSTANTS.C_MAX_RULES] OF ST_User_Rule;

    // Sensor calibration pipeline
    G_Calib_Outdoor_Temp : ST_Sensor_Calibration_Record;
    G_Calib_Ambient_Lux : ST_Sensor_Calibration_Record;
    G_Calib_Supply_Temps : ARRAY[1..GVL_CONSTANTS.C_MAX_SUPPLY_TEMPS] OF ST_Sensor_Calibration_Record;
    G_Calib_Room_Temps : ARRAY[1..GVL_CONSTANTS.C_MAX_ZONES] OF ST_Sensor_Calibration_Record;
    G_Calib_Floor_Temps : ARRAY[1..GVL_CONSTANTS.C_MAX_ZONES] OF ST_Sensor_Calibration_Record;
    G_Calib_CO2 : ARRAY[1..GVL_CONSTANTS.C_MAX_ZONES] OF ST_Sensor_Calibration_Record;
    G_Calib_Humidity : ARRAY[1..GVL_CONSTANTS.C_MAX_ZONES] OF ST_Sensor_Calibration_Record;
    G_Calib_Manifold_T_Supply : ARRAY[1..GVL_CONSTANTS.C_MAX_MANIFOLDS] OF ST_Sensor_Calibration_Record;
    G_Calib_Manifold_T_Return : ARRAY[1..GVL_CONSTANTS.C_MAX_MANIFOLDS] OF ST_Sensor_Calibration_Record;
    G_Calib_Methane : ARRAY[1..GVL_CONSTANTS.C_MAX_METHANE_SENSORS] OF ST_Sensor_Calibration_Record;
    G_Calib_CO : ARRAY[1..GVL_CONSTANTS.C_MAX_CO_SENSORS] OF ST_Sensor_Calibration_Record;

    // Valve test configuration
    G_Valve_Test_Config : ARRAY[1..GVL_CONSTANTS.C_MAX_MANIFOLDS] OF ST_Valve_Test_Config;

    // HMI Commands & States
    G_HMI_Apply_Settings : BOOL;
    G_HMI_Mute_Alarm : BOOL;
    G_HMI_Ack_Alarms : BOOL;

    // Entrance lighting assist configuration.
    // Physical lux connection is optional and can be enabled later from HMI/config.
    G_Entrance_Light_Assist_Enabled : BOOL := TRUE;
    G_Entrance_Light_Assist_Use_Lux_Sensor : BOOL := FALSE;
    G_Entrance_Light_Assist_Fallback_To_Night : BOOL := TRUE;
    G_Entrance_Light_Assist_Lux_Threshold : REAL := 50.0;
    G_Entrance_Light_Assist_Duration_MS : UDINT := 300000;
    G_Entrance_Door_1_Index : INT := 1;
    G_Entrance_Door_2_Index : INT := 2;
    G_Entrance_Corridor_Light_Zone : INT := 1;
    G_Entrance_Stairs_Light_Zone : INT := 2;
    G_Entrance_Corridor_Light_Level : BYTE := 100;
    G_Entrance_Stairs_Light_Level : BYTE := 30;

    // Access Control Commands
    G_HMI_Gate_Open_Req : BOOL;
    G_HMI_Wicket_Open_Req : BOOL;
    G_HMI_Lock_1_Open_Req : BOOL;
    G_HMI_Lock_1_Close_Req : BOOL;
    G_HMI_Lock_2_Open_Req : BOOL;
    G_HMI_Lock_2_Close_Req : BOOL;
    G_Access_Pulse_MS : UDINT := 500;

    // Network security
    G_Allowed_IPs : ARRAY[1..GVL_CONSTANTS.C_MAX_ALLOWED_IPS] OF STRING(15) := ['192.168.1.100','192.168.1.101','127.0.0.1','',''];

    G_Backup_Circulation_Pump_In_Service : BOOL := TRUE;
    G_Electric_Heater_In_Service : BOOL := TRUE;
    G_Freeze_Hardware_Retry_Count : INT := 2;
    G_Freeze_Hardware_Retry_Delay_MS : UDINT := 5000;
    G_Pump_Exercise_Enabled : BOOL := TRUE;
    G_Pump_Exercise_Interval_MS : UDINT := 604800000;
    G_Pump_Exercise_Duration_MS : UDINT := 30000;
    G_Manifold_Pump_In_Service : ARRAY[1..GVL_CONSTANTS.C_MAX_MANIFOLDS] OF BOOL := [TRUE, TRUE, TRUE, TRUE, TRUE];
    G_Manifold_Priority : ARRAY[1..GVL_CONSTANTS.C_MAX_MANIFOLDS] OF INT := [3, 3, 2, 2, 1];
    G_Manifold_Thermal_Weight : ARRAY[1..GVL_CONSTANTS.C_MAX_MANIFOLDS] OF REAL := [1.0, 1.0, 0.8, 0.8, 0.5];
    G_Max_Active_Manifolds : INT := 3;
    G_Max_Thermal_Budget : REAL := 6.0;
    G_Policy_Min_Hold_MS : UDINT := 300000;
    G_DHW_Heating_Pump_In_Service : BOOL := TRUE;
    G_DHW_Circ_Pump_In_Service : BOOL := TRUE;
    G_Water_Valve_Exercise_Enabled : BOOL := TRUE;
    G_Water_Valve_Exercise_Interval_MS : UDINT := 604800000;
    G_Water_Valve_Exercise_Duration_MS : UDINT := 15000;
    G_Water_Valve_Close_Retry_Count : INT := 2;
    G_Water_Valve_Close_Retry_Delay_MS : UDINT := 3000;

    // OpenTherm / Modbus adapter configuration
    G_OpenTherm_Enabled : BOOL := FALSE;
    G_OpenTherm_Heartbeat_Timeout_MS : UDINT := 5000;
    G_OpenTherm_Command_Ack_Timeout_MS : UDINT := 3000;
    G_OpenTherm_Register_Map : ARRAY[1..GVL_CONSTANTS.C_MAX_BOILERS] OF ST_OpenTherm_Register_Map;

    // Modbus RTU transport configuration
    // Scalar fields are used instead of nested structure for CODESYS/build-system compatibility.
    G_Modbus_RTU_Driver_Attached : BOOL := FALSE;
    G_Modbus_RTU_Port_Number : BYTE := 1; // 1=COM1, 2=COM2, 3=COM3, 4=COM4
    G_Modbus_RTU_Baudrate : UDINT := 9600;
    G_Modbus_RTU_Parity : BYTE := 1; // 0=None, 1=Even, 2=Odd
    G_Modbus_RTU_Stop_Bits : BYTE := 1; // 1 or 2
    G_Modbus_RTU_Data_Bits : BYTE := 8; // usually 8
    G_Modbus_RTU_Slave_ID : BYTE := 1;
    G_Modbus_RTU_Poll_Interval_MS : UDINT := 100;
    G_Modbus_RTU_Request_Timeout_MS : UDINT := 250;
    G_Modbus_RTU_Retry_Count : INT := 2;

    // IO Mapping
    G_FloorTemp_Map : ARRAY[1..GVL_CONSTANTS.C_MAX_HEATING_CIRCUITS] OF INT := [1, 2, 3, 4, 5, 6, 7, 8, 9, 10, 11, 12, 13, 14, 15, 16];
    G_RoomTemp_Map : ARRAY[1..16] OF INT := [1, 2, 3, 4, 5, 6, 7, 8, 9, 10, 11, 12, 13, 14, 15, 16];
    G_Door_Map : ARRAY[1..GVL_CONSTANTS.C_MAX_DOOR_SENSORS] OF INT := [1, 2, 3, 4, 5, 6, 7, 8];
    G_Window_Map : ARRAY[1..16] OF INT := [9, 10, 11, 12, 13, 14, 15, 16, 17, 18, 19, 20, 21, 22, 23, 24];

    // Evacuation config
    C_MAX_LIGHT_ZONES : INT := 32;
    G_Evac_Exit_Zones : ARRAY[1..32] OF BOOL;
    G_Evac_Zone_Names : ARRAY[1..32] OF STRING(80);

END_VAR

VAR_GLOBAL CONSTANT
    C_MS_PER_SEC : UDINT := GVL_CONSTANTS.C_MS_IN_SECOND;
    C_SEC_PER_MIN : UDINT := 60;
    C_MIN_PER_HOUR : UDINT := 60;
    C_MS_PER_MIN : UDINT := GVL_CONSTANTS.C_MS_IN_MINUTE;
    C_MAX_RULES : INT := 20;
    C_ZONE_COUNT : BYTE := 18;

    ERR_PRESSURE_OUT_OF_RANGE : UDINT := 16#E004;
    ERR_HIGH_DELTA_T : UDINT := 16#E005;
    ERR_BOILER_OFFLINE : UDINT := 16#E006;
    ERR_BOILER_GENERAL_FAULT : UDINT := 16#E007;
    ERR_BOILER_NO_FLAME : UDINT := 16#E008;
    ERR_PUMP_NO_CURRENT : UDINT := 16#E009;
    ERR_PUMP_UNDERCURRENT : UDINT := 16#E00A;
    ERR_PUMP_OVERCURRENT : UDINT := 16#E00B;
    ERR_DELTA_T_LOW : UDINT := 16#E00C;
    ERR_DELTA_T_HIGH : UDINT := 16#E00D;
    ERR_DHW_IO_OFFLINE : UDINT := 16#E00E;
    ERR_DHW_TEMP_SENSOR_FAULT : UDINT := 16#E00F;
    ERR_DHW_PRESSURE_OUT_OF_RANGE : UDINT := 16#E010;
    ERR_DHW_PRESSURE_SENSOR_FAULT : UDINT := 16#E011;
    ERR_BACKUP_PUMP_OUT_OF_SERVICE : UDINT := 16#E012;
    ERR_ELECTRIC_HEATER_OUT_OF_SERVICE : UDINT := 16#E013;
    ERR_MANIFOLD_PUMP_OUT_OF_SERVICE : UDINT := 16#E014;
    ERR_DHW_HEATING_PUMP_OUT_OF_SERVICE : UDINT := 16#E015;
    ERR_DHW_CIRC_PUMP_OUT_OF_SERVICE : UDINT := 16#E016;
    ERR_FREEZE_HARDWARE_FAILED : UDINT := 16#E017;
END_VAR

(* ---- GVL_Config_Activation.gvl ---- *)
{attribute 'qualified_only'}
VAR_GLOBAL RETAIN
    G_Requested_Config_Version : UDINT;
    G_Staged_Config_Version : UDINT;
    G_Last_Stable_Config_Version : UDINT;

    G_Activation_Request : BOOL;
    G_Rollback_Request : BOOL;
END_VAR

VAR_GLOBAL
    G_Staged_Topology_Config : ARRAY[1..64] OF ST_Water_Topology_Config_Record;

    G_Activation_State : ST_Config_Activation_State;

    G_Config_Quarantine_Active : BOOL;
    G_Activation_Runtime_Valid : BOOL;
    G_Last_Update_MS : UDINT;

    G_Status_Code : UINT;
    G_Status_Text : STRING(160);
END_VAR

(* ---- GVL_CONTROL_TIMING_FABRIC.gvl ---- *)
VAR_GLOBAL
    // Global deterministic control-loop timing authority.
    Control_Temporal_Coherence_Valid : BOOL := FALSE;
    Control_Temporal_Coherence_Granted : BOOL := FALSE;
    Control_Temporal_Coherence_Quarantine_Active : BOOL := TRUE;

    // Deterministic temporal coherence proofs.
    Loop_Sampling_Coherent : BOOL := FALSE;
    Feedback_Freshness_Valid : BOOL := FALSE;
    PID_Phase_Alignment_Valid : BOOL := FALSE;
    Cross_Loop_Temporal_Stable : BOOL := FALSE;
    Multi_Rate_Causality_Coherent : BOOL := FALSE;

    // Timing-window validators.
    Control_Snapshot_Epoch_Coherent : BOOL := FALSE;
    Feedback_Window_Stable : BOOL := FALSE;
    Loop_Execution_Phase_Stable : BOOL := FALSE;
    Temporal_Observation_Aligned : BOOL := FALSE;

    // Temporal aliasing / oscillation detectors.
    PID_Phase_Skew_Detected : BOOL := FALSE;
    Sampling_Window_Divergence_Detected : BOOL := FALSE;
    Feedback_Freshness_Aliasing_Detected : BOOL := FALSE;
    Cross_Loop_Stabilization_Lag_Detected : BOOL := FALSE;
    Multi_Rate_Oscillation_Risk_Detected : BOOL := FALSE;
    Distributed_Control_Ringing_Detected : BOOL := FALSE;

    // Control timing epochs.
    Control_Timing_Epoch : UDINT := 0;
    Control_Timing_Epoch_Coherent : BOOL := FALSE;

    // Temporal authority.
    Control_Timing_Last_Update_MS : UDINT := 0;
    Control_Timing_Lease_Expired : BOOL := TRUE;

    // Diagnostics.
    Control_Timing_Last_Error_Code : UDINT := 0;
    Control_Timing_Last_Error_Text : STRING(160) := '';
    Control_Timing_Invalidation_Count : UDINT := 0;
END_VAR

(* ---- GVL_DEGRADED.gvl ---- *)
VAR_GLOBAL
    G_System_Degraded : BOOL := FALSE;
    G_Degraded_Mode_Active : BOOL := FALSE;
    G_Degraded_Recovery_Required : BOOL := FALSE;
END_VAR

(* ---- GVL_DISTRIBUTED_COMMIT.gvl ---- *)
VAR_GLOBAL
    // ======================================================
    // DISTRIBUTED PUBLICATION COMMIT STATE
    // ======================================================
    // Deterministic peer publication commit handshake foundation.
    // Publication-continuity governance only.
    // Does not invalidate runtime barrier, PLC fencing
    // or local immutable snapshot authority.
    // ======================================================

    Distributed_Commit_Epoch : ULINT := 0;
    Distributed_Commit_Reconciliation_Epoch : ULINT := 0;

    Local_Publication_Commit_Epoch : ULINT := 0;
    Peer_Publication_Commit_Epoch : ULINT := 0;

    Local_Prepare_Epoch : ULINT := 0;
    Peer_Prepare_Epoch : ULINT := 0;

    Publication_Prepare_Active : BOOL := FALSE;
    Publication_Prepare_Valid : BOOL := FALSE;
    Publication_Commit_Requested : BOOL := FALSE;
    Publication_Commit_Confirmed : BOOL := FALSE;

    Peer_Commit_Ack_Valid : BOOL := FALSE;
    Peer_Commit_Ack_Expired : BOOL := FALSE;
    Peer_Commit_Mismatch : BOOL := FALSE;
    Peer_Commit_Replay_Detected : BOOL := FALSE;
    Peer_Commit_Missing : BOOL := FALSE;

    Commit_Lease_Active : BOOL := FALSE;
    Commit_Lease_Expired : BOOL := FALSE;
    Commit_Timeout_MS : UDINT := 5000;

    Local_Commit_Last_Refresh_MS : UDINT := 0;
    Peer_Commit_Last_Refresh_MS : UDINT := 0;
    Commit_Last_Reconciliation_MS : UDINT := 0;

    Distributed_Commit_Valid : BOOL := FALSE;
    Distributed_Commit_Quarantine_Active : BOOL := FALSE;

    Distributed_Commit_Last_Error_Code : UDINT := 0;
    Distributed_Commit_Last_Error_Text : STRING(160) := '';
END_VAR

(* ---- GVL_DISTRIBUTED_EPOCH_LINEARITY_FABRIC.gvl ---- *)
VAR_GLOBAL
    Distributed_Epoch_Linearity_Valid : BOOL := FALSE;
    Distributed_Epoch_Linearity_Granted : BOOL := FALSE;

    Distributed_Epoch_Linearity_Valid_Proof : BOOL := FALSE;
    Epoch_Timeline_Monotonic : BOOL := FALSE;
    Cluster_Epoch_Consensus_Stable : BOOL := FALSE;

    Epoch_Causality_Grounded : BOOL := FALSE;
    Distributed_Epoch_Lineage_Coherent : BOOL := FALSE;

    Epoch_Rollback_Detected : BOOL := FALSE;
    Distributed_Epoch_Fork_Detected : BOOL := FALSE;
    Stale_Epoch_Application_Detected : BOOL := FALSE;

    Distributed_Epoch_Linearity_Epoch : UDINT := 0;
END_VAR

(* ---- GVL_Distributed_Execution_Gates.gvl ---- *)
{attribute 'qualified_only'}
VAR_GLOBAL
    G_Can_Replicate : BOOL;
    G_Can_Execute : BOOL;
    G_Can_Orchestrate : BOOL;
    G_Can_Recover : BOOL;
    G_Can_Rollback : BOOL;
    G_Can_Own_Projection : BOOL;

    G_Runtime_Valid : BOOL;
    G_Last_Update_MS : UDINT;

    G_Status_Code : UINT;
    G_Status_Text : STRING(160);
END_VAR

(* ---- GVL_Distributed_Recovery_Lock.gvl ---- *)
VAR_GLOBAL
    G_Recovery_Lock : ST_Distributed_Recovery_Lock;

    G_Runtime_Valid : BOOL := FALSE;
    G_Last_Update_MS : UDINT := 0;

    G_Recovery_Execution_Blocked : BOOL := TRUE;
    G_Rollback_Execution_Blocked : BOOL := TRUE;
    G_Reopen_Execution_Blocked : BOOL := TRUE;

    G_Status_Code : UINT := 0;
    G_Status_Text : STRING(160) := '';
END_VAR

(* ---- GVL_DOMAIN_EXECUTION_POLICY.gvl ---- *)
{attribute 'qualified_only'}
VAR_GLOBAL
    // Domain execution policy. Observational first layer.
    // This GVL classifies when a domain needs critical, periodic or idle execution.
    // It does not directly control physical outputs.
    // Mode convention: 0 = idle, 1 = periodic, 2 = critical.

    G_Last_Update_MS : UDINT := 0;

    // Scenario/context classification.
    G_Security_Context_Active : BOOL := FALSE;
    G_Away_Context_Active : BOOL := FALSE;
    G_Presence_Context_Active : BOOL := FALSE;
    G_Emergency_Context_Active : BOOL := FALSE;

    // Periodic observation intervals.
    Access_Periodic_Interval_MS : UDINT := 1000;
    Lighting_Periodic_Interval_MS : UDINT := 1000;
    Water_Periodic_Interval_MS : UDINT := 1000;
    Heating_Periodic_Interval_MS : UDINT := 5000;
    Vent_Periodic_Interval_MS : UDINT := 3000;
    Simulation_Periodic_Interval_MS : UDINT := 1000;

    // Access.
    Access_Mode : UINT := 0;
    Access_Critical_Run : BOOL := FALSE;
    Access_Periodic_Run : BOOL := FALSE;
    Access_Periodic_Due : BOOL := FALSE;
    Access_Idle_By_Design : BOOL := FALSE;

    // Lighting.
    Lighting_Mode : UINT := 0;
    Lighting_Critical_Run : BOOL := FALSE;
    Lighting_Periodic_Run : BOOL := FALSE;
    Lighting_Periodic_Due : BOOL := FALSE;
    Lighting_Idle_By_Design : BOOL := FALSE;

    // Water.
    Water_Mode : UINT := 0;
    Water_Critical_Run : BOOL := FALSE;
    Water_Periodic_Run : BOOL := FALSE;
    Water_Periodic_Due : BOOL := FALSE;
    Water_Idle_By_Design : BOOL := FALSE;

    // Heating.
    Heating_Mode : UINT := 0;
    Heating_Critical_Run : BOOL := FALSE;
    Heating_Periodic_Run : BOOL := FALSE;
    Heating_Periodic_Due : BOOL := FALSE;
    Heating_Idle_By_Design : BOOL := FALSE;

    // Ventilation.
    Vent_Mode : UINT := 0;
    Vent_Critical_Run : BOOL := FALSE;
    Vent_Periodic_Run : BOOL := FALSE;
    Vent_Periodic_Due : BOOL := FALSE;
    Vent_Idle_By_Design : BOOL := FALSE;

    // Simulation.
    Simulation_Mode : UINT := 0;
    Simulation_Context_Active : BOOL := FALSE;
    Simulation_Run_Allowed : BOOL := FALSE;
    Simulation_Periodic_Due : BOOL := FALSE;
    Simulation_Idle_By_Design : BOOL := FALSE;

    // Summary.
    Any_Critical_Run : BOOL := FALSE;
    Any_Periodic_Run : BOOL := FALSE;
    Any_Periodic_Due : BOOL := FALSE;
    Any_Idle_By_Design : BOOL := FALSE;
    Status_Code : UINT := 0;
    Status_Text : STRING(160) := '';
END_VAR

(* ---- GVL_ENERGY_CAUSALITY_FABRIC.gvl ---- *)
VAR_GLOBAL
    // Global deterministic energy causality authority.
    Energy_Causality_Valid : BOOL := FALSE;
    Energy_Causality_Granted : BOOL := FALSE;
    Energy_Causality_Quarantine_Active : BOOL := TRUE;

    // Energetic realizability proofs.
    Hydraulic_Energy_State_Valid : BOOL := FALSE;
    Thermal_Energy_State_Valid : BOOL := FALSE;
    Electrical_Load_State_Valid : BOOL := FALSE;
    Motor_Energy_Envelope_Valid : BOOL := FALSE;
    Distributed_Load_Coherent : BOOL := FALSE;

    // Stable plant energy envelopes.
    Energy_Envelope_Stable : BOOL := FALSE;
    Transient_Load_Stable : BOOL := FALSE;
    Thermal_Accumulation_Stable : BOOL := FALSE;
    Recovery_Energy_Coherent : BOOL := FALSE;

    // Energy divergence detectors.
    DryRun_Energy_State_Detected : BOOL := FALSE;
    Thermal_Extraction_Divergence_Detected : BOOL := FALSE;
    Load_Synchronization_Spike_Detected : BOOL := FALSE;
    Hydraulic_Energy_Starvation_Detected : BOOL := FALSE;
    Distributed_Transient_Overload_Detected : BOOL := FALSE;
    Energy_Recovery_Instability_Detected : BOOL := FALSE;

    // Energy authority epochs.
    Energy_Causality_Epoch : UDINT := 0;
    Energy_Causality_Epoch_Coherent : BOOL := FALSE;

    // Temporal authority.
    Energy_Causality_Last_Update_MS : UDINT := 0;
    Energy_Causality_Lease_Expired : BOOL := TRUE;

    // Diagnostics.
    Energy_Causality_Last_Error_Code : UDINT := 0;
    Energy_Causality_Last_Error_Text : STRING(160) := '';
    Energy_Causality_Invalidation_Count : UDINT := 0;
END_VAR

(* ---- GVL_ENERGY_RESURRECTION_BOUNDARY_FABRIC.gvl ---- *)
VAR_GLOBAL
    Energy_Resurrection_Boundary_Valid : BOOL := FALSE;
    Energy_Resurrection_Boundary_Granted : BOOL := FALSE;

    Energy_Resurrection_Causality_Valid : BOOL := FALSE;
    Energy_Authority_Recovery_Bounded : BOOL := FALSE;
    CrossDomain_Energy_Recovery_Stable : BOOL := FALSE;

    Energy_Resurrection_Ordering_Valid : BOOL := FALSE;
    Distributed_Energy_Recovery_Consensus : BOOL := FALSE;

    Unsafe_Energy_Resurrection_Detected : BOOL := FALSE;
    CrossDomain_Energy_Recovery_Race : BOOL := FALSE;
    Energy_Recovery_Fork_Detected : BOOL := FALSE;

    Energy_Resurrection_Epoch : UDINT := 0;
END_VAR

(* ---- GVL_GOVERNANCE_FEEDBACK_INTEGRITY_FABRIC.gvl ---- *)
VAR_GLOBAL
    // Deterministic governance feedback integrity governance.
    Governance_Feedback_Integrity_Valid : BOOL := FALSE;
    Governance_Feedback_Integrity_Granted : BOOL := FALSE;
    Governance_Feedback_Integrity_Quarantine_Active : BOOL := TRUE;

    // Governance feedback causality proofs.
    Execution_Feedback_Causality_Isolated : BOOL := FALSE;
    Governance_Derivation_Inputs_Canonical : BOOL := FALSE;
    Telemetry_To_Authority_Lineage_Valid : BOOL := FALSE;
    Feedback_Epoch_Integrity_Stable : BOOL := FALSE;
    Governance_Feedback_Lineage_Coherent : BOOL := FALSE;

    // Feedback integrity validation.
    Authenticated_Execution_Observation_Valid : BOOL := FALSE;
    CrossEpoch_Feedback_Continuity_Stable : BOOL := FALSE;
    Governance_Input_Causality_Grounded : BOOL := FALSE;
    Distributed_Feedback_Consensus_Valid : BOOL := FALSE;

    // Governance feedback poisoning detectors.
    Governance_Feedback_Poisoning_Detected : BOOL := FALSE;
    Execution_Telemetry_Authority_Corruption : BOOL := FALSE;
    CrossEpoch_Feedback_Lineage_Drift : BOOL := FALSE;
    Retroactive_Governance_Mutation_Detected : BOOL := FALSE;
    Distributed_Feedback_Fork_Detected : BOOL := FALSE;
    Untrusted_Execution_Observation_Injected : BOOL := FALSE;

    // Feedback epochs.
    Governance_Feedback_Integrity_Epoch : UDINT := 0;
    Governance_Feedback_Integrity_Epoch_Coherent : BOOL := FALSE;

    // Temporal authority.
    Governance_Feedback_Integrity_Last_Update_MS : UDINT := 0;
    Governance_Feedback_Integrity_Lease_Expired : BOOL := TRUE;

    // Diagnostics.
    Governance_Feedback_Integrity_Last_Error_Code : UDINT := 0;
    Governance_Feedback_Integrity_Last_Error_Text : STRING(160) := '';
    Governance_Feedback_Integrity_Invalidation_Count : UDINT := 0;
END_VAR

(* ---- GVL_GOVERNANCE_PUBLICATION_BINDING_FABRIC.gvl ---- *)
VAR_GLOBAL
    // Deterministic governance publication binding governance.
    Governance_Publication_Binding_Valid : BOOL := FALSE;
    Governance_Publication_Binding_Granted : BOOL := FALSE;
    Governance_Publication_Binding_Quarantine_Active : BOOL := TRUE;

    // Observability publication binding proofs.
    Observability_Publication_Causality_Valid : BOOL := FALSE;
    Upstream_Governance_Lease_Fresh : BOOL := FALSE;
    Governance_Publication_Epoch_Coherent : BOOL := FALSE;
    Publication_Quarantine_Propagation_Valid : BOOL := FALSE;
    Canonical_Observability_Reality_Consistent : BOOL := FALSE;

    // Publication integrity validation.
    Diagnostics_Publication_Consistency_Valid : BOOL := FALSE;
    HMI_Publication_State_Aligned : BOOL := FALSE;
    Blackbox_Invalidation_Lineage_Valid : BOOL := FALSE;
    Distributed_Publication_Consensus_Valid : BOOL := FALSE;

    // Stale-valid publication detectors.
    Stale_Valid_Publication_Detected : BOOL := FALSE;
    LeaseExpired_Governance_Published_As_Healthy : BOOL := FALSE;
    Quarantine_State_Publication_Bypass : BOOL := FALSE;
    Governance_Invalidation_Hidden_From_Observability : BOOL := FALSE;
    Distributed_Publication_State_Fork_Detected : BOOL := FALSE;
    Historical_Invalidation_Causality_Lost : BOOL := FALSE;

    // Publication epochs.
    Governance_Publication_Binding_Epoch : UDINT := 0;
    Governance_Publication_Binding_Epoch_Coherent_Runtime : BOOL := FALSE;

    // Temporal authority.
    Governance_Publication_Binding_Last_Update_MS : UDINT := 0;
    Governance_Publication_Binding_Lease_Expired : BOOL := TRUE;

    // Diagnostics.
    Governance_Publication_Binding_Last_Error_Code : UDINT := 0;
    Governance_Publication_Binding_Last_Error_Text : STRING(160) := '';
    Governance_Publication_Binding_Invalidation_Count : UDINT := 0;
END_VAR

(* ---- GVL_GOVERNANCE_VALIDATOR_INTEGRITY_FABRIC.gvl ---- *)
VAR_GLOBAL
    // Deterministic governance validator integrity governance.
    Governance_Validator_Integrity_Valid : BOOL := FALSE;
    Governance_Validator_Integrity_Granted : BOOL := FALSE;
    Governance_Validator_Integrity_Quarantine_Active : BOOL := TRUE;

    // Validator immutability proofs.
    Validator_Semantics_Immutable : BOOL := FALSE;
    CrossEpoch_Validation_Equivalence_Stable : BOOL := FALSE;
    Distributed_Validator_Consensus_Valid : BOOL := FALSE;
    Governance_Rule_Integrity_Canonical : BOOL := FALSE;
    Validator_Lineage_Coherent : BOOL := FALSE;

    // Validator integrity validation.
    Validator_Causality_Grounded : BOOL := FALSE;
    Governance_Rule_Evolution_Governed : BOOL := FALSE;
    Distributed_Validation_Timeline_Monotonic : BOOL := FALSE;
    Validator_Interpretation_Equivalence_Valid : BOOL := FALSE;

    // Validator self-corruption detectors.
    Validator_Semantic_Drift_Detected : BOOL := FALSE;
    CrossNode_Validation_Fork : BOOL := FALSE;
    Governance_Rule_Mutation_Detected : BOOL := FALSE;
    SelfReferential_Validator_Corruption : BOOL := FALSE;
    Validator_Lineage_Drift_Detected : BOOL := FALSE;
    Distributed_Validator_Reality_Fork_Detected : BOOL := FALSE;

    // Validator epochs.
    Governance_Validator_Integrity_Epoch : UDINT := 0;
    Governance_Validator_Integrity_Epoch_Coherent : BOOL := FALSE;

    // Temporal authority.
    Governance_Validator_Integrity_Last_Update_MS : UDINT := 0;
    Governance_Validator_Integrity_Lease_Expired : BOOL := TRUE;

    // Diagnostics.
    Governance_Validator_Integrity_Last_Error_Code : UDINT := 0;
    Governance_Validator_Integrity_Last_Error_Text : STRING(160) := '';
    Governance_Validator_Integrity_Invalidation_Count : UDINT := 0;
END_VAR

(* ---- GVL_HEATING_DIAGNOSTICS.gvl ---- *)
VAR_GLOBAL
    G_Manifold_Pressure_Fault : ARRAY[1..16] OF BOOL;
    G_Manifold_Current_Fault : ARRAY[1..16] OF BOOL;
    G_Manifold_Return_Temp_Fault : ARRAY[1..16] OF BOOL;
END_VAR

(* ---- GVL_HEATING_POLICY.gvl ---- *)
{attribute 'qualified_only'}
VAR_GLOBAL
    G_Zone_Empty_Duration_MS : ARRAY[1..GVL_CONSTANTS.C_MAX_ZONES] OF UDINT;
    G_Zone_Permanent_Use : ARRAY[1..GVL_CONSTANTS.C_MAX_ZONES] OF BOOL;
    G_Zone_Guest_Preheat_Request : ARRAY[1..GVL_CONSTANTS.C_MAX_ZONES] OF BOOL;
    G_Zone_Policy_Class : ARRAY[1..GVL_CONSTANTS.C_MAX_ZONES] OF INT;
    G_Zone_Target_Adjustment : ARRAY[1..GVL_CONSTANTS.C_MAX_ZONES] OF REAL;
    G_Zone_Priority_Bias : ARRAY[1..GVL_CONSTANTS.C_MAX_ZONES] OF REAL;

    G_Policy_Mode : E_Heating_Policy_Mode := E_Heating_Policy_Mode.HPM_NORMAL;
    G_Policy_Block_Heating_Request : BOOL;
    G_Policy_Target_Adjustment : REAL;
    G_Policy_Priority_Multiplier : REAL := 1.0;
    G_Policy_Self_Tune_Active : BOOL;
    G_Policy_Self_Tune_Level : INT;
    G_Policy_Feedback_Stable : BOOL;
    G_Policy_Feedback_Improving : BOOL;
    G_Policy_Feedback_Quality : REAL;
    G_Policy_Predictive_Active : BOOL;
    G_Policy_Predictive_Adjustment : REAL;

    // zone intelligence
    G_Zone_Quality : ARRAY[1..GVL_CONSTANTS.C_MAX_ZONES] OF REAL;
    G_Zone_Improving : ARRAY[1..GVL_CONSTANTS.C_MAX_ZONES] OF BOOL;
    G_Zone_Stable : ARRAY[1..GVL_CONSTANTS.C_MAX_ZONES] OF BOOL;
    G_Zone_Self_Level : ARRAY[1..GVL_CONSTANTS.C_MAX_ZONES] OF INT;

    // thermal model: 1.0 = normal inertia, >1 slower/heavier, <1 faster/lighter
    G_Zone_Thermal_Inertia : ARRAY[1..GVL_CONSTANTS.C_MAX_ZONES] OF REAL := [1.0, 1.0, 1.0, 1.0, 1.0, 1.0, 1.0, 1.0, 1.0, 1.0, 1.0, 1.0, 1.0, 1.0, 1.0, 1.0];
    G_Zone_Thermal_Response : ARRAY[1..GVL_CONSTANTS.C_MAX_ZONES] OF REAL;
    G_Zone_Thermal_Demand : ARRAY[1..GVL_CONSTANTS.C_MAX_ZONES] OF REAL;
    G_Zone_Time_To_Heat_MS : ARRAY[1..GVL_CONSTANTS.C_MAX_ZONES] OF UDINT;
    G_Zone_Preheat_Needed : ARRAY[1..GVL_CONSTANTS.C_MAX_ZONES] OF BOOL;

    // thermal model v2 diagnostics
    G_Zone_Heat_Loss_Rate : ARRAY[1..GVL_CONSTANTS.C_MAX_ZONES] OF REAL;
    G_Zone_Heat_Gain_Rate : ARRAY[1..GVL_CONSTANTS.C_MAX_ZONES] OF REAL;
    G_Zone_Predicted_Temp_30m : ARRAY[1..GVL_CONSTANTS.C_MAX_ZONES] OF REAL;
    G_Zone_Thermal_Model_Confidence : ARRAY[1..GVL_CONSTANTS.C_MAX_ZONES] OF REAL;

    // optimization diagnostics
    G_Zone_Optimization_Score : ARRAY[1..GVL_CONSTANTS.C_MAX_ZONES] OF REAL;
    G_Optimization_Load_Index : REAL;
    G_Optimization_Energy_Saving_Active : BOOL;

    // schedule-aware preheat. Comfort time is milliseconds from midnight.
    G_Zone_Schedule_Enabled : ARRAY[1..GVL_CONSTANTS.C_MAX_ZONES] OF BOOL;
    G_Zone_Comfort_Time_MS : ARRAY[1..GVL_CONSTANTS.C_MAX_ZONES] OF UDINT;
    G_Zone_Schedule_Preheat_Active : ARRAY[1..GVL_CONSTANTS.C_MAX_ZONES] OF BOOL;
    G_Zone_Schedule_Learned_Offset_MS : ARRAY[1..GVL_CONSTANTS.C_MAX_ZONES, 1..3] OF UDINT;
END_VAR

(* ---- GVL_Heating_Source_Stability.gvl ---- *)
{attribute 'qualified_only'}
VAR_GLOBAL
    // Predictive source-stability observability layer.
    // Observation-only: no runtime authority, no valve ownership,
    // no direct influence on heating outputs.

    // Canonical predictive observability contract.
    G_State : ARRAY[1..GVL_CONSTANTS.C_MAX_HEATING_CIRCUITS] OF ST_Heating_Runtime_Source_Instability_State;
END_VAR

(* ---- GVL_HISTORICAL_TRUTH.gvl ---- *)
VAR_GLOBAL
    // Global immutable historical truth authority.
    Historical_Truth_Valid : BOOL := FALSE;
    Historical_Truth_Granted : BOOL := FALSE;
    Historical_Truth_Quarantine_Active : BOOL := TRUE;

    // Immutable causality proofs.
    Trend_History_Causally_Immutable : BOOL := FALSE;
    Alarm_Chronology_Immutable : BOOL := FALSE;
    Blackbox_Snapshot_Immutable : BOOL := FALSE;
    Diagnostics_History_Coherent : BOOL := FALSE;
    Failover_Chronology_Coherent : BOOL := FALSE;

    // Historical persistence integrity.
    Persisted_Epochs_Coherent : BOOL := FALSE;
    Recovery_Replay_Coherent : BOOL := FALSE;
    Historical_Snapshot_Coherent : BOOL := FALSE;
    Mixed_Authority_Persistence_Absent : BOOL := FALSE;

    // Historical corruption detectors.
    History_Epoch_Skew_Detected : BOOL := FALSE;
    Failover_Chronology_Corruption_Detected : BOOL := FALSE;
    Trend_Replay_Race_Detected : BOOL := FALSE;
    Blackbox_Causality_Drift_Detected : BOOL := FALSE;
    Alarm_Order_Reconstruction_Error : BOOL := FALSE;
    Mixed_Authority_Persistence_Detected : BOOL := FALSE;

    // Historical authority epochs.
    Historical_Truth_Epoch : UDINT := 0;
    Historical_Truth_Epoch_Coherent : BOOL := FALSE;

    // Temporal historical authority.
    Historical_Last_Update_MS : UDINT := 0;
    Historical_Lease_Expired : BOOL := TRUE;

    // Diagnostics.
    Historical_Last_Error_Code : UDINT := 0;
    Historical_Last_Error_Text : STRING(160) := '';
    Historical_Invalidation_Count : UDINT := 0;
END_VAR

(* ---- GVL_INTENT_POLICY.gvl ---- *)
{attribute 'qualified_only'}
VAR_GLOBAL
    // Policy intent signals (NO logic, only transport)

    G_Preheat_Request : BOOL;
    G_Freeze_Request : BOOL;

    // Zone-level intents
    G_Zone_Target_Adjustment : ARRAY[1..GVL_CONSTANTS.C_MAX_ZONES] OF REAL;

END_VAR

(* ---- GVL_INTENT_SYSTEM.gvl ---- *)
VAR_GLOBAL
    // --- meta ---
    I_Source_Valid : BOOL := FALSE;
    I_Last_Update_Cycle : UDINT := 0;
    I_Last_Update_MS : UDINT := 0;

    // --- system mode constraints ---
    I_Mode_Safe_Stop_Active : BOOL := FALSE;
    I_Mode_Degraded_Active : BOOL := FALSE;
    I_Mode_Freeze_Protection_Active : BOOL := FALSE;

    // --- scenario / automation ---
    I_Preheat_Request : BOOL := FALSE;
    I_Freeze_Request : BOOL := FALSE;
    I_Scenario_Request_Allowed : BOOL := FALSE;
    I_Operator_Scenario_Block : BOOL := FALSE;

    // --- gateway / system permissions ---
    I_Gateway_Command_Valid : BOOL := FALSE;
    I_Gateway_Command_Type : INT := 0;
    I_Gateway_Writes_Allowed : BOOL := FALSE;
    I_Reset_Errors_Request : BOOL := FALSE;
    I_Config_Apply_Allowed : BOOL := FALSE;
    I_Time_Sync_Allowed : BOOL := FALSE;
    I_Temperature_Write_Allowed : BOOL := FALSE;
    I_Ventilation_Write_Allowed : BOOL := FALSE;
    I_Maintenance_Apply_Allowed : BOOL := FALSE;

    // --- command gate block flags ---
    I_Lighting_Overrides_Block : BOOL := FALSE;
    I_Blinds_Overrides_Block : BOOL := FALSE;
    I_Socket_Overrides_Block : BOOL := FALSE;

    // --- permissions / constraints ---
    I_Access_Open_Allowed : BOOL := FALSE;
    I_Manual_Override_Allowed : BOOL := FALSE;
    I_Dangerous_Action_Allowed : BOOL := FALSE;
END_VAR

(* ---- GVL_IO.gvl ---- *)
{attribute 'qualified_only'}
VAR_GLOBAL
    // ======================================================
    // PHYSICAL IO SURFACE
    // ======================================================
    // Input fields are hardware/mapping observations.
    // Output fields are the terminal physical publication surface.
    //
    // PRG_IO_Write is the only runtime-layer publisher for physical
    // output commands in this GVL. Upstream authority/governance,
    // verifier, recovery and observability layers must not write
    // physical outputs directly.
    // ======================================================

    DI_Security_Open : ARRAY[1..GVL_CONSTANTS.C_MAX_SECURITY_SENSORS] OF BOOL;
    DI_Security_Glass : ARRAY[1..GVL_CONSTANTS.C_MAX_SECURITY_SENSORS] OF BOOL;
    DI_Security_2F_Group : BOOL;
    DI_Flood_Sensors : ARRAY[1..GVL_CONSTANTS.C_MAX_FLOOD_SENSORS] OF BOOL;
    DI_Manifold_End_Switches : ARRAY[1..GVL_CONSTANTS.C_MAX_MANIFOLDS] OF BOOL;
    AO_Manifold_Valves : ARRAY[1..GVL_CONSTANTS.C_MAX_MANIFOLDS] OF UINT;
    DO_Manifold_Pumps : ARRAY[1..GVL_CONSTANTS.C_MAX_MANIFOLDS] OF BOOL;
    AI_Manifold_Currents : ARRAY[1..GVL_CONSTANTS.C_MAX_MANIFOLDS] OF INT;
    AI_Manifold_Pressures : ARRAY[1..GVL_CONSTANTS.C_MAX_MANIFOLDS] OF INT;
    AI_Manifold_Temps_Supply : ARRAY[1..GVL_CONSTANTS.C_MAX_MANIFOLDS] OF ST_Owen_Analog_Value;
    AI_Manifold_Temps_Return : ARRAY[1..GVL_CONSTANTS.C_MAX_MANIFOLDS] OF INT;
    AO_Supply_Fans : ARRAY[1..GVL_CONSTANTS.C_MAX_SUPPLY_FANS] OF UINT;
    AO_Exhaust_Fans : ARRAY[1..GVL_CONSTANTS.C_MAX_EXHAUST_FANS] OF UINT;
    AO_Lighting_Levels : ARRAY[1..GVL_CONSTANTS.C_MAX_LIGHT_ZONES] OF UINT;
    AO_Blinds_Positions : ARRAY[1..GVL_CONSTANTS.C_MAX_BLINDS] OF UINT;
    AI_Supply_Temps : ARRAY[1..GVL_CONSTANTS.C_MAX_SUPPLY_TEMPS] OF ST_Owen_Analog_Value;
    AI_Boiler_Modulation : ARRAY[1..GVL_CONSTANTS.C_MAX_BOILERS] OF INT;
    AI_Boiler_Flame_Status : ARRAY[1..GVL_CONSTANTS.C_MAX_BOILERS] OF BOOL;
    DI_Boiler_Error : ARRAY[1..GVL_CONSTANTS.C_MAX_BOILERS] OF BOOL;
    AI_Methane_LEL : ARRAY[1..GVL_CONSTANTS.C_MAX_METHANE_SENSORS] OF ST_Owen_Analog_Value;
    AI_CO_PPM : ARRAY[1..GVL_CONSTANTS.C_MAX_CO_SENSORS] OF REAL;
    DI_Smoke_Sensors : ARRAY[1..GVL_CONSTANTS.C_MAX_SMOKE_SENSORS] OF BOOL;
    AI_Temp_Outdoor : ST_Owen_Analog_Value;
    AI_Ambient_Lux : ST_Owen_Analog_Value;
    AI_Floor_Temps : ARRAY[1..GVL_CONSTANTS.C_MAX_ZONES] OF REAL;
    AI_Room_Temps : ARRAY[1..GVL_CONSTANTS.C_MAX_ZONES] OF REAL;
    AI_Room_Hum : ARRAY[1..GVL_CONSTANTS.C_MAX_ZONES] OF REAL;
    AI_Room_CO2 : ARRAY[1..GVL_CONSTANTS.C_MAX_ZONES] OF REAL;
    DO_Zone_Valves : ARRAY[1..GVL_CONSTANTS.C_MAX_HEATING_CIRCUITS] OF BOOL;
    AI_DHW_Temp : REAL;
    AI_DHW_Pressure : REAL;
    DO_DHW_Heating_Pump : BOOL;
    DO_DHW_Circ_Pump : BOOL;
    DO_Backup_Circulation_Pump : BOOL;
    DO_Electric_Heater_Enable : BOOL;
    DI_Lighting_Switches : ARRAY[1..GVL_CONSTANTS.C_MAX_LIGHT_ZONES] OF BOOL;
    DI_Socket_Switches : ARRAY[1..GVL_CONSTANTS.C_MAX_SOCKETS] OF BOOL;
    DI_Motion_Sensors : ARRAY[1..GVL_CONSTANTS.C_MAX_LIGHT_ZONES] OF BOOL;
    DO_Sockets : ARRAY[1..GVL_CONSTANTS.C_MAX_SOCKETS] OF BOOL;
    DO_Gas_Valve_Close : BOOL;

    // Water common inlet valves: 35 = ХВС, 36 = ГВС.
    DO_Water_Valve_35_Open : BOOL;
    DO_Water_Valve_35_Close : BOOL;
    DO_Water_Valve_36_Open : BOOL;
    DO_Water_Valve_36_Close : BOOL;

    // Water local riser valves: 1/2 riser 1, 3/4 riser 2, 5/6 riser 3.
    DO_Water_Local_Valve_Open : ARRAY[1..6] OF BOOL;
    DO_Water_Local_Valve_Close : ARRAY[1..6] OF BOOL;

    AI_Water_Valve_35_Current : REAL;
    AI_Water_Valve_36_Current : REAL;
    DI_Power_OK : BOOL;
    DO_Gas_Siren : BOOL;
    DO_Fire_Siren : BOOL;
    DO_Security_Siren : BOOL;
    DO_Pump_Main_Enable : BOOL;
    DO_Gate_Open : BOOL;
    DO_Wicket_Open : BOOL;
    DO_Lock_1_Open : BOOL;
    DO_Lock_1_Close : BOOL;
    DO_Lock_2_Open : BOOL;
    DO_Lock_2_Close : BOOL;
    DI_Partner_Pulse : BOOL;
    DI_Partner_Active : BOOL;
    DO_Heartbeat_Pulse : BOOL;
    DO_Active_Status : BOOL;
    DI_Module_1_Heartbeat : BOOL;
    DI_Module_2_Heartbeat : BOOL;
    DI_Backup_Circulation_Pump_Feedback : BOOL;
    DI_Electric_Heater_Feedback : BOOL;
    DI_Water_Zone_Open_FB : ARRAY[1..GVL_CONSTANTS.C_MAX_WATER_ZONES] OF BOOL;
    DI_Water_Zone_Close_FB : ARRAY[1..GVL_CONSTANTS.C_MAX_WATER_ZONES] OF BOOL;
    DO_Water_Zone_Enable : ARRAY[1..GVL_CONSTANTS.C_MAX_WATER_ZONES] OF BOOL;
END_VAR

(* ---- GVL_IO_WRITE_RUNTIME_BUFFER.gvl ---- *)
{attribute 'qualified_only'}
VAR_GLOBAL
    // Runtime buffer owned by PRG_IO_Write and its phase programs only.

    B_Heating_Forced_Off : BOOL := FALSE;
    B_Vent_Forced_Off : BOOL := FALSE;
    B_Water_Forced_Off : BOOL := FALSE;
    B_Access_Forced_Off : BOOL := FALSE;
    B_Access_Safety_Override : BOOL := FALSE;

    B_Global_Hard_Stop : BOOL := FALSE;
    B_Gas_Safety_Stop : BOOL := FALSE;
    B_Freeze_Active : BOOL := FALSE;

    B_PreOutput_Block_IO : BOOL := FALSE;
    B_Output_Freshness_Block : BOOL := FALSE;
    B_Output_Publication_Block : BOOL := FALSE;
    B_Distributed_Publication_Block : BOOL := FALSE;
    B_Snapshot_Block : BOOL := FALSE;
    B_Distributed_Execution_Block : BOOL := FALSE;

    B_Gas_Fire_Siren_Enable : BOOL := FALSE;
    B_Gas_Siren_Authority : BOOL := FALSE;
    B_Fire_Siren_Authority : BOOL := FALSE;
END_VAR

(* ---- GVL_LIGHTING_RUNTIME.gvl ---- *)
{attribute 'qualified_only'}
VAR_GLOBAL
    // Lighting domain execution feedback. Observational only.

    G_Runtime_Required : BOOL := FALSE;
    G_Runtime_Executed : BOOL := FALSE;
    G_Runtime_Idle_By_Design : BOOL := FALSE;
    G_Runtime_Blocked_By_Distributed_Gates : BOOL := FALSE;
    G_Emergency_Override_Active : BOOL := FALSE;
    G_Any_Light_Active : BOOL := FALSE;
    G_Any_Blind_Not_Safe_Open : BOOL := FALSE;
    G_Any_Socket_Active : BOOL := FALSE;
    G_Last_Update_MS : UDINT := 0;
    G_Status_Code : UINT := 0;
    G_Status_Text : STRING(128) := '';
END_VAR

(* ---- GVL_LIGHTING_RUNTIME_BUFFER.gvl ---- *)
{attribute 'qualified_only'}
VAR_GLOBAL
    // Runtime buffer owned by PRG_Lighting and its phase programs only.

    B_Manual_Light_Override : ARRAY[1..GVL_CONSTANTS.C_MAX_LIGHT_ZONES] OF BYTE;
    B_Manual_Blinds_Override : ARRAY[1..GVL_CONSTANTS.C_MAX_LIGHT_ZONES] OF BYTE;
    B_Manual_Socket_Override : ARRAY[1..GVL_CONSTANTS.C_MAX_SOCKETS] OF BOOL;

    B_Sim_Lights : ARRAY[1..GVL_CONSTANTS.C_MAX_LIGHT_ZONES] OF BOOL;
    B_Physical_Switches : ARRAY[1..GVL_CONSTANTS.C_MAX_LIGHT_ZONES] OF BOOL;
    B_Motion_Sensors : ARRAY[1..GVL_CONSTANTS.C_MAX_LIGHT_ZONES] OF BOOL;
    B_Blinds_Override : ARRAY[1..GVL_CONSTANTS.C_MAX_BLINDS] OF BYTE;
    B_Socket_Override : ARRAY[1..GVL_CONSTANTS.C_MAX_SOCKETS] OF BOOL;
    B_Wet_Zone_Light_Active : ARRAY[1..GVL_CONSTANTS.C_MAX_WET_ZONES] OF BOOL;

    B_Fire_Alarm_Active : BOOL := FALSE;
    B_Flood_Alarm_Active : BOOL := FALSE;
    B_Security_Armed : BOOL := FALSE;
    B_Security_Alarm : BOOL := FALSE;
    B_Evac_Blink_On : BOOL := FALSE;

    B_Distributed_Execute_Allowed : BOOL := FALSE;
    B_Distributed_Projection_Allowed : BOOL := FALSE;
    B_Emergency_Lighting_Override : BOOL := FALSE;
END_VAR

(* ---- GVL_MODBUS_SCAN.gvl ---- *)
{attribute 'qualified_only'}
VAR_GLOBAL
    // ======================================================
    // SAFE READ-ONLY MODBUS REGISTER SCAN
    // ======================================================
    // This scanner NEVER writes registers.
    // Only FC03/FC04 are allowed.

    G_Scan_Enable : BOOL := FALSE;
    G_Scan_Active : BOOL := FALSE;
    G_Scan_Done : BOOL := FALSE;
    G_Scan_Error : BOOL := FALSE;

    G_Slave_ID : BYTE := 1;

    G_Start_Register : UINT := 0;
    G_End_Register : UINT := 255;
    G_Current_Register : UINT := 0;

    G_Found_Register : ARRAY[0..255] OF BOOL;
    G_Found_Value : ARRAY[0..255] OF WORD;

    G_Last_Scan_MS : UDINT := 0;
END_VAR

(* ---- GVL_MODE.gvl ---- *)
{attribute 'qualified_only'}
VAR_GLOBAL
    G_Current_Behavior_Mode : E_Behavior_Mode := BEHAVIOR_HOME;
    G_Mode_Last_Change_TS : UDINT := 0;
    G_Mode_Code : UDINT := 0;

    // Explicit behavior-mode requests
    G_Away_Request : BOOL := FALSE;
    G_Maintenance_Request : BOOL := FALSE;
END_VAR

(* ---- GVL_OBSERVABILITY_TRUTH.gvl ---- *)
VAR_GLOBAL
    // Global observability truth authority.
    Observability_Truth_Valid : BOOL := FALSE;
    Observability_Truth_Granted : BOOL := FALSE;
    Observability_Truth_Quarantine_Active : BOOL := TRUE;

    // Authoritative operator visibility.
    HMI_Authority_Coherent : BOOL := FALSE;
    Alarm_Authority_Coherent : BOOL := FALSE;
    Trend_Authority_Coherent : BOOL := FALSE;
    Diagnostics_Authority_Coherent : BOOL := FALSE;
    History_Authority_Coherent : BOOL := FALSE;

    // Projection causality.
    HMI_Epoch_Coherent : BOOL := FALSE;
    Alarm_Publication_Coherent : BOOL := FALSE;
    Trend_Causality_Coherent : BOOL := FALSE;
    Diagnostics_Causality_Coherent : BOOL := FALSE;
    Operator_Visibility_Consistent : BOOL := FALSE;

    // Observability split-brain detection.
    Stale_HMI_Epoch_Detected : BOOL := FALSE;
    Alarm_Publication_Lag_Detected : BOOL := FALSE;
    Trend_Causality_Skew_Detected : BOOL := FALSE;
    Diagnostic_Truth_Race_Detected : BOOL := FALSE;
    Operator_Visibility_Fragmentation_Detected : BOOL := FALSE;
    Authority_UI_Divergence_Detected : BOOL := FALSE;

    // Observability authority epochs.
    Observability_Truth_Epoch : UDINT := 0;
    Observability_Truth_Epoch_Coherent : BOOL := FALSE;

    // Temporal observability authority.
    Observability_Last_Update_MS : UDINT := 0;
    Observability_Lease_Expired : BOOL := TRUE;

    // Diagnostics.
    Observability_Last_Error_Code : UDINT := 0;
    Observability_Last_Error_Text : STRING(160) := '';
    Observability_Invalidation_Count : UDINT := 0;
END_VAR

(* ---- GVL_OPENTHERM_ADAPTER.gvl ---- *)
{attribute 'qualified_only'}
VAR_GLOBAL
    // ======================================================
    // PHYSICAL OPENTHERM ADAPTER RUNTIME STATE
    // ======================================================
    // Static transport configuration lives in GVL_CONFIG.
    // This GVL contains runtime command/status/wire image only.

    G_Command : ARRAY[1..GVL_CONSTANTS.C_MAX_BOILERS] OF ST_OpenTherm_Command;
    G_Status : ARRAY[1..GVL_CONSTANTS.C_MAX_BOILERS] OF ST_OpenTherm_Status;

    // Raw wire image exchanged with transport layer
    G_Wire_Image : ARRAY[1..GVL_CONSTANTS.C_MAX_BOILERS] OF ST_OpenTherm_Wire_Image;

    // Transport diagnostics
    G_Transport_Online : BOOL := FALSE;
    G_Transport_Error : BOOL := FALSE;
    G_Last_Transport_Update_MS : UDINT := 0;
END_VAR

(* ---- GVL_OPERATOR_SEMANTIC_ALIGNMENT.gvl ---- *)
VAR_GLOBAL
    // Global deterministic operator semantic alignment authority.
    Operator_Semantic_Alignment_Valid : BOOL := FALSE;
    Operator_Semantic_Alignment_Granted : BOOL := FALSE;
    Operator_Semantic_Alignment_Quarantine_Active : BOOL := TRUE;

    // Human-machine semantic coherence proofs.
    HMI_Semantic_State_Coherent : BOOL := FALSE;
    Operator_Recovery_Intent_Aligned : BOOL := FALSE;
    Alarm_Semantic_Priority_Coherent : BOOL := FALSE;
    Runtime_Explanation_Coherent : BOOL := FALSE;
    Authority_State_Human_Visible : BOOL := FALSE;

    // Operator cognition synchronization.
    Human_Interpretation_Coherent : BOOL := FALSE;
    Adaptive_Runtime_Visibility_Valid : BOOL := FALSE;
    Semantic_Explanation_Fresh : BOOL := FALSE;
    Operator_Action_Context_Aligned : BOOL := FALSE;

    // Human-machine semantic split-brain detectors.
    HMI_Semantic_Lag_Detected : BOOL := FALSE;
    Operator_Interpretation_Skew_Detected : BOOL := FALSE;
    Alarm_Cognition_Mismatch_Detected : BOOL := FALSE;
    Hidden_Authority_State_Detected : BOOL := FALSE;
    Semantic_Explanation_Divergence_Detected : BOOL := FALSE;
    Human_Recovery_Misunderstanding_Detected : BOOL := FALSE;

    // Alignment epochs.
    Operator_Alignment_Epoch : UDINT := 0;
    Operator_Alignment_Epoch_Coherent : BOOL := FALSE;

    // Temporal authority.
    Operator_Alignment_Last_Update_MS : UDINT := 0;
    Operator_Alignment_Lease_Expired : BOOL := TRUE;

    // Diagnostics.
    Operator_Alignment_Last_Error_Code : UDINT := 0;
    Operator_Alignment_Last_Error_Text : STRING(160) := '';
    Operator_Alignment_Invalidation_Count : UDINT := 0;
END_VAR

(* ---- GVL_OUTDOOR_LIGHTING.gvl ---- *)
{attribute 'qualified_only'}
VAR_GLOBAL
    // ======================================================
    // OUTDOOR LIGHTING / LANDSCAPE CONFIG + RUNTIME SURFACE
    // ======================================================
    // Logical outdoor zones are mapped to existing lighting/socket domains.
    // No direct physical IO writes are performed here.
    // Physical module/channel mapping is a porting-stage task.
    // ======================================================

    // Global enable and darkness source.
    G_Outdoor_Enabled : BOOL := TRUE;
    G_Outdoor_Use_Lux_Sensor : BOOL := FALSE;
    G_Outdoor_Fallback_To_Night : BOOL := TRUE;
    G_Outdoor_Lux_Threshold : REAL := 50.0;

    // Logical mappings. Defaults reserve the tail of lighting/socket arrays.
    // 1=paths, 2=facade, 3=trees/shrubs, 4=architectural/perimeter.
    G_Outdoor_Light_Zone_Index : ARRAY[1..GVL_CONSTANTS.C_MAX_OUTDOOR_ZONES] OF INT := [29, 30, 31, 32];
    G_Outdoor_Motion_Zone_Index : ARRAY[1..GVL_CONSTANTS.C_MAX_OUTDOOR_ZONES] OF INT := [29, 30, 31, 32];
    G_Outdoor_Socket_Index : ARRAY[1..GVL_CONSTANTS.C_MAX_OUTDOOR_ZONES] OF INT := [33, 34, 35, 36];

    // Light levels by mode.
    G_Outdoor_Auto_Level : BYTE := 40;
    G_Outdoor_Economy_Level : BYTE := 10;
    G_Outdoor_Party_Level : BYTE := 100;
    G_Outdoor_Security_Level : BYTE := 80;

    // Economy window, default 23:00-06:00.
    G_Outdoor_Economy_Start_MS : UDINT := 82800000;
    G_Outdoor_Economy_End_MS : UDINT := 21600000;

    // Landscape socket policy.
    G_Outdoor_Sockets_Enabled : BOOL := TRUE;
    G_Outdoor_Sockets_On_In_Party : BOOL := TRUE;
    G_Outdoor_Sockets_On_In_Auto : BOOL := FALSE;
    G_Outdoor_Sockets_Off_In_Security : BOOL := TRUE;

    // Per-zone manual override from HMI/gateway.
    G_Outdoor_Manual_Mode : ARRAY[1..GVL_CONSTANTS.C_MAX_OUTDOOR_ZONES] OF BOOL;
    G_Outdoor_Manual_Light_Level : ARRAY[1..GVL_CONSTANTS.C_MAX_OUTDOOR_ZONES] OF BYTE;
    G_Outdoor_Manual_Socket_State : ARRAY[1..GVL_CONSTANTS.C_MAX_OUTDOOR_ZONES] OF BOOL;

    // Runtime status.
    G_Outdoor_Dark_Active : BOOL;
    G_Outdoor_Economy_Active : BOOL;
    G_Outdoor_Party_Active : BOOL;
    G_Outdoor_Security_Active : BOOL;
    G_Outdoor_Light_Level : ARRAY[1..GVL_CONSTANTS.C_MAX_OUTDOOR_ZONES] OF BYTE;
    G_Outdoor_Socket_State : ARRAY[1..GVL_CONSTANTS.C_MAX_OUTDOOR_ZONES] OF BOOL;
    G_Outdoor_Status_Text : STRING(200) := 'OUTDOOR DISABLED';
END_VAR

(* ---- GVL_OUTPUT_EPOCH.gvl ---- *)
VAR_GLOBAL
    // ======================================================
    // OUTPUT PUBLICATION AUTHORITY STATE
    // ======================================================
    // Centralized final physical publication arbitration state.
    // ======================================================

    Output_Publication_Epoch : ULINT := 0;
    Output_Publication_Valid : BOOL := FALSE;
    Output_Publication_Allowed : BOOL := TRUE;

    Output_Lease_Active : BOOL := FALSE;
    Output_Lease_Expired : BOOL := FALSE;
    Output_Lease_Timeout_MS : UDINT := 3000;

    Output_Last_Publication_MS : UDINT := 0;
    Output_Last_Refresh_MS : UDINT := 0;
    Output_Last_Invalidation_MS : UDINT := 0;

    Output_Runtime_Epoch : ULINT := 0;
    Output_Runtime_Epoch_Valid : BOOL := FALSE;

    Output_Stale_Detected : BOOL := FALSE;
    Output_Forced_Safe_Decay : BOOL := FALSE;

    Output_Semantic_Continuity_Warning : BOOL := FALSE;

    Output_Last_Error_Code : UDINT := 0;
    Output_Last_Error_Text : STRING(160) := '';
END_VAR

(* ---- GVL_PASSIVE_RUNTIME_VERIFICATION_FABRIC.gvl ---- *)
VAR_GLOBAL
    Passive_Runtime_Verification_Active : BOOL := TRUE;

    Runtime_Verification_Consistency_Valid : BOOL := FALSE;
    Runtime_Verification_Lineage_Coherent : BOOL := FALSE;
    Runtime_Verification_Timeline_Monotonic : BOOL := FALSE;

    Passive_Runtime_Verification_ReadOnly : BOOL := TRUE;
    Passive_Runtime_Verification_NoMutation : BOOL := TRUE;
    Passive_Runtime_Verification_NoAuthority : BOOL := TRUE;
    Passive_Runtime_Verification_NoBlocking : BOOL := TRUE;

    Runtime_Semantic_Drift_Observed : BOOL := FALSE;
    Runtime_Consistency_Decay_Observed : BOOL := FALSE;
    Runtime_Verification_Anomaly_Observed : BOOL := FALSE;

    Passive_Runtime_Verification_Epoch : UDINT := 0;
END_VAR

(* ---- GVL_PHYSICAL_AUTHORITY_EPOCH.gvl ---- *)
VAR_GLOBAL
    // Global physical authority epoch.
    Physical_Authority_Epoch : UDINT := 0;
    Physical_Authority_Epoch_Valid : BOOL := FALSE;

    // Cross-governor epoch coherence.
    Snapshot_Epoch_Coherent : BOOL := FALSE;
    Consensus_Epoch_Coherent : BOOL := FALSE;
    Causality_Epoch_Coherent : BOOL := FALSE;
    PreOutput_Epoch_Coherent : BOOL := FALSE;

    // Epoch divergence detection.
    Physical_Epoch_Drift_Detected : BOOL := FALSE;
    Physical_Epoch_Replay_Suspected : BOOL := FALSE;
    Partial_Epoch_Advancement_Detected : BOOL := FALSE;
    Cross_Cycle_Epoch_Skew_Detected : BOOL := FALSE;

    // Temporal authority.
    Physical_Authority_Lease_Expired : BOOL := TRUE;
    Physical_Authority_Quarantine_Active : BOOL := TRUE;
    Physical_Authority_Last_Update_MS : UDINT := 0;

    // Diagnostics.
    Physical_Authority_Last_Error_Code : UDINT := 0;
    Physical_Authority_Last_Error_Text : STRING(160) := '';
    Physical_Authority_Invalidation_Count : UDINT := 0;
END_VAR

(* ---- GVL_PHYSICAL_SAFESTATE_LATTICE_FABRIC.gvl ---- *)
VAR_GLOBAL
    // Deterministic physical safe-state lattice governance.
    Physical_SafeState_Lattice_Valid : BOOL := FALSE;
    Physical_SafeState_Lattice_Granted : BOOL := FALSE;
    Physical_SafeState_Lattice_Quarantine_Active : BOOL := TRUE;

    // Canonical safe-state topology proofs.
    Canonical_SafeState_Topology_Valid : BOOL := FALSE;
    Physical_SafeState_Lattice_Coherent : BOOL := FALSE;
    Deterministic_FailSafe_Convergence_Granted : BOOL := FALSE;
    SafeState_Energy_Boundary_Stable : BOOL := FALSE;
    SafeState_Physical_Risk_Bounded : BOOL := FALSE;

    // Domain safe-state compatibility.
    Heating_SafeState_Compatible : BOOL := FALSE;
    Water_SafeState_Compatible : BOOL := FALSE;
    Ventilation_SafeState_Compatible : BOOL := FALSE;
    Access_SafeState_Compatible : BOOL := FALSE;
    Lighting_SafeState_Compatible : BOOL := FALSE;

    // Physical safe-state convergence validators.
    Thermal_SafeState_Stable : BOOL := FALSE;
    Hydraulic_SafeState_Stable : BOOL := FALSE;
    Airflow_SafeState_Stable : BOOL := FALSE;
    Occupancy_SafeState_Stable : BOOL := FALSE;
    Residual_Actuation_Safe : BOOL := FALSE;

    // Safe-state ambiguity detectors.
    SafeState_Ambiguity_Detected : BOOL := FALSE;
    Partial_SafeState_Asymmetry_Detected : BOOL := FALSE;
    Physical_SafeState_Deadlock_Detected : BOOL := FALSE;
    Unsafe_SafeState_Topology_Detected : BOOL := FALSE;
    Residual_Unsafe_Actuation_Detected : BOOL := FALSE;
    SafeState_Energy_Leakage_Detected : BOOL := FALSE;

    // Safe-state epochs.
    Physical_SafeState_Lattice_Epoch : UDINT := 0;
    Physical_SafeState_Lattice_Epoch_Coherent : BOOL := FALSE;

    // Temporal authority.
    Physical_SafeState_Lattice_Last_Update_MS : UDINT := 0;
    Physical_SafeState_Lattice_Lease_Expired : BOOL := TRUE;

    // Diagnostics.
    Physical_SafeState_Lattice_Last_Error_Code : UDINT := 0;
    Physical_SafeState_Lattice_Last_Error_Text : STRING(160) := '';
    Physical_SafeState_Lattice_Invalidation_Count : UDINT := 0;
END_VAR

(* ---- GVL_PLC_FENCING.gvl ---- *)
VAR_GLOBAL
    // ======================================================
    // DISTRIBUTED PLC OWNERSHIP / FENCING STATE
    // ======================================================
    // Centralized ownership epoch governance.
    // Used to prevent split-brain and stale-owner resurrection.
    // ======================================================

    PLC_Ownership_Epoch : ULINT := 0;
    PLC_Fencing_Token : ULINT := 0;

    PLC_Ownership_Valid : BOOL := FALSE;
    PLC_Semantic_Authority_Valid : BOOL := FALSE;
    PLC_Heartbeat_Only_Mode : BOOL := FALSE;

    PLC_Lease_Active : BOOL := FALSE;
    PLC_Lease_Expired : BOOL := FALSE;
    PLC_Lease_Timeout_MS : UDINT := 5000;

    PLC_Last_Lease_Refresh_MS : UDINT := 0;
    PLC_Last_Authority_Validation_MS : UDINT := 0;

    PLC_Split_Brain_Detected : BOOL := FALSE;
    PLC_Stale_Owner_Detected : BOOL := FALSE;
    PLC_Asymmetric_Partition_Detected : BOOL := FALSE;

    PLC_Forced_Safe_Quarantine : BOOL := FALSE;

    PLC_Last_Error_Code : UDINT := 0;
    PLC_Last_Error_Text : STRING(160) := '';

    PLC_Fencing_Invalidation_Count : UDINT := 0;
END_VAR

(* ---- GVL_RECOVERY_REACTIVATION_CONTROL_FABRIC.gvl ---- *)
VAR_GLOBAL
    Recovery_Reactivation_Control_Valid : BOOL := FALSE;
    Recovery_Reactivation_Control_Granted : BOOL := FALSE;

    Recovery_Reactivation_Boundary_Stable : BOOL := FALSE;
    CrossSubsystem_Reactivation_Consistent : BOOL := FALSE;
    Reactivation_Energy_Boundary_Safe : BOOL := FALSE;

    Reactivation_Causality_Grounded : BOOL := FALSE;
    Reactivation_Ordering_Stable : BOOL := FALSE;

    Unsafe_Reactivation_Ordering_Detected : BOOL := FALSE;
    Partial_Reactivation_Leak_Detected : BOOL := FALSE;
    CrossSubsystem_Reactivation_Fork : BOOL := FALSE;

    Recovery_Reactivation_Epoch : UDINT := 0;
END_VAR

(* ---- GVL_RESIDUAL_ENERGY_STATE_FABRIC.gvl ---- *)
VAR_GLOBAL
    Residual_Energy_State_Valid : BOOL := FALSE;
    Residual_Energy_Bounded : BOOL := FALSE;
    Residual_Actuation_Energy_Safe : BOOL := FALSE;
    Thermal_Energy_Dissipation_Stable : BOOL := FALSE;

    Residual_Energy_Causality_Valid : BOOL := FALSE;
    Distributed_Residual_Energy_Consensus : BOOL := FALSE;

    Latent_Unsafe_Actuation_Detected : BOOL := FALSE;
    Residual_Energy_Persistence_Detected : BOOL := FALSE;
    Unsafe_Thermal_Energy_Retention : BOOL := FALSE;

    Residual_Energy_Epoch : UDINT := 0;
END_VAR

(* ---- GVL_RUNTIME_ASSUMPTION_INTEGRITY_FABRIC.gvl ---- *)
VAR_GLOBAL
    Runtime_Assumption_Integrity_Active : BOOL := TRUE;

    Runtime_Assumption_Integrity_Observed : BOOL := FALSE;
    Runtime_Assumption_Lineage_Coherent : BOOL := FALSE;
    Runtime_Assumption_Stability_Observed : BOOL := FALSE;

    Runtime_Assumption_ReadOnly_Mode : BOOL := TRUE;
    Runtime_Assumption_NoAuthorityMutation : BOOL := TRUE;

    Runtime_Assumption_Decay_Observed : BOOL := FALSE;
    Runtime_Assumption_Violation_Observed : BOOL := FALSE;
    Runtime_Assumption_Drift_Observed : BOOL := FALSE;

    Runtime_Assumption_Integrity_Epoch : UDINT := 0;
END_VAR

(* ---- GVL_RUNTIME_IO_VALIDATION.gvl ---- *)
{attribute 'qualified_only'}
VAR_GLOBAL
    G_Last_Update_MS : UDINT := 0;
    G_Validation_Executed : BOOL := FALSE;
    G_Validation_Valid : BOOL := TRUE;

    Fire_IO_Valid : BOOL := TRUE;
    Gas_IO_Valid : BOOL := TRUE;
    Leak_IO_Valid : BOOL := TRUE;
    Global_Stop_IO_Valid : BOOL := TRUE;
    Inactive_PLC_IO_Valid : BOOL := TRUE;
    Freeze_IO_Valid : BOOL := TRUE;

    Any_IO_Invalid : BOOL := FALSE;
    Status_Code : UINT := 0;
    Status_Text : STRING(160) := '';
END_VAR

(* ---- GVL_SAFETY_OBSERVABILITY_TRUTH_FABRIC.gvl ---- *)
VAR_GLOBAL
    Safety_Observability_Truth_Valid : BOOL := FALSE;
    Safety_Observability_Truth_Granted : BOOL := FALSE;

    Safety_Reality_Projection_Valid : BOOL := FALSE;
    Observability_Reality_Equivalence_Granted : BOOL := FALSE;
    Safety_Projection_Causality_Grounded : BOOL := FALSE;
    Physical_Safety_Projection_Canonical : BOOL := FALSE;

    Distributed_Safety_Projection_Consensus : BOOL := FALSE;
    Safety_Observability_Lineage_Coherent : BOOL := FALSE;

    FakeSafe_Projection_Detected : BOOL := FALSE;
    Telemetry_Reality_Divergence_Detected : BOOL := FALSE;
    Stale_Safety_Projection_Detected : BOOL := FALSE;
    Safety_Observability_Fork_Detected : BOOL := FALSE;

    Safety_Observability_Epoch : UDINT := 0;
END_VAR

(* ---- GVL_SEMANTIC_PROGRESS.gvl ---- *)
VAR_GLOBAL
    // ======================================================
    // SEMANTIC PROGRESS CONTINUITY STATE
    // ======================================================
    // Isolated semantic execution continuity foundation.
    // Visibility/publication continuity only.
    // Does not directly invalidate runtime barrier,
    // PLC fencing, immutable snapshots or IO authority.
    //
    // This surface tracks real runtime phase evidence so
    // semantic progress is no longer self-counter-only.
    // ======================================================

    Semantic_Progress_Epoch : ULINT := 0;
    Semantic_Continuity_Epoch : ULINT := 0;

    Semantic_Forward_Progress_Valid : BOOL := FALSE;
    Semantic_Execution_Continuity_OK : BOOL := FALSE;

    Semantic_Execution_Counter : ULINT := 0;
    Semantic_Last_Execution_Counter : ULINT := 0;

    Semantic_Progress_Last_Update_MS : UDINT := 0;
    Semantic_Progress_Timeout_MS : UDINT := 10000;

    Semantic_Stagnation_Detected : BOOL := FALSE;
    Semantic_Replay_Suspected : BOOL := FALSE;
    Semantic_Livelock_Suspected : BOOL := FALSE;
    Semantic_Deadlock_Suspected : BOOL := FALSE;

    Semantic_Progress_Lease_Active : BOOL := FALSE;
    Semantic_Progress_Lease_Expired : BOOL := FALSE;

    Semantic_Progress_Quarantine_Active : BOOL := FALSE;

    // ------------------------------------------------------
    // Runtime phase evidence observed by semantic governor.
    // ------------------------------------------------------
    Semantic_Runtime_Barrier_Epoch : ULINT := 0;
    Semantic_Runtime_Snapshot_Epoch : ULINT := 0;
    Semantic_Distributed_Commit_Epoch : ULINT := 0;
    Semantic_Output_Publication_Epoch : ULINT := 0;

    Semantic_Last_Runtime_Barrier_Epoch : ULINT := 0;
    Semantic_Last_Runtime_Snapshot_Epoch : ULINT := 0;
    Semantic_Last_Distributed_Commit_Epoch : ULINT := 0;
    Semantic_Last_Output_Publication_Epoch : ULINT := 0;

    Semantic_Runtime_Barrier_Evidence_OK : BOOL := FALSE;
    Semantic_Runtime_Snapshot_Evidence_OK : BOOL := FALSE;
    Semantic_Distributed_Commit_Evidence_OK : BOOL := FALSE;
    Semantic_Output_Publication_Evidence_OK : BOOL := FALSE;

    Semantic_Phase_Evidence_OK : BOOL := FALSE;
    Semantic_Phase_Stall_Detected : BOOL := FALSE;
    Semantic_Output_Stall_Detected : BOOL := FALSE;

    Semantic_Last_Error_Code : UDINT := 0;
    Semantic_Last_Error_Text : STRING(160) := '';

    Semantic_Invalidation_Count : UDINT := 0;
END_VAR
